KUKA KRL program: EPS_2_251806_MH02A_A_20260213065129.src

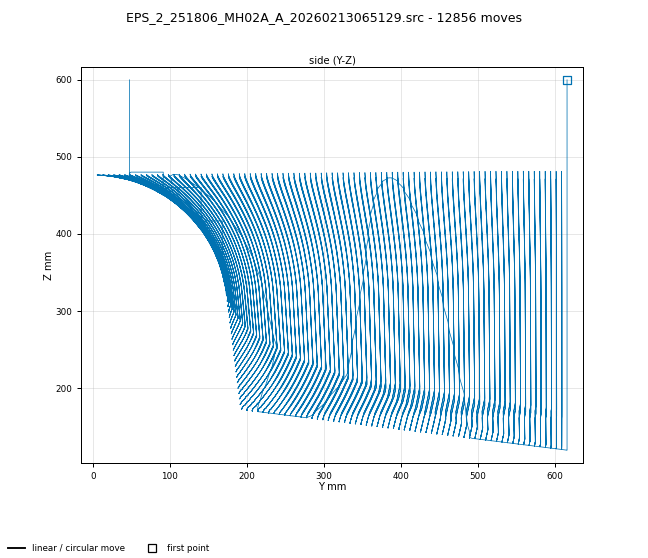
[picture p0: tool path of EPS_2_251806_MH02A_A_20260213065129.src, 12856 of 12858 moves have a stored position in this frame; points joined in program order, loops and branches not executed]
&ACCESS RVP
&REL 4
&COMMENT QRS 19112012
&PARAM EDITMASK = *
DEF PART()
EXT BAS (BAS_COMMAND :IN,REAL :IN )
INT I
BAS (#INITMOV,0 )

;KUKA QRS Post kuka4.cps  Date:22-06-2017 !

File_ID=3031

QRS_PRE_INIT()

;Init var - Until changes are made in qrs_pre_init
Outlet_Square_prg=0
Inlet_1_Square_prg=0
Inlet_2_Square_prg=0
Inlet_3_Square_prg=0
Inlet_4_Square_prg=0
Inlet_5_Square_prg=0

Outlet_1={X 0.000, Y 534.640, Z 332.000, B 0.000, E1 0.000 }
Inlet_1={X 0.000, Y 535.370, Z 322.000, B 0.000, E1 180.000 }
Outlet_1_type=299
Inlet_1_type=299
;QRS#1=Sidecore dimensions
;QRS#2=300-12" PVC SDR 35
;QRS#3=300-12" PVC SDR 35
;QRS#4=
;QRS#5=
;QRS#6=
;QRS#7=
;QRS#8=
;QRS#9=16M PSX
;QRS#10=16M PSX
;QRS#11=
;QRS#12=
;QRS#13=
;QRS#14=
;QRS#15=
;QRS#16=1220x127x762 2,5'
;QRS#17=EPS Height
;QRS#18=481,5
;QRS#19=*
;QRS#20= UPDATED VERSION 22-06-2017
;QRS#21=*
Outlet_Square=0150
Inlet_1_Square=0150
Inlet_2_Square=0
Inlet_3_Square=0
Inlet_4_Square=0
Inlet_5_Square=0
Mill_Square=1
Outlet_Square_Prg=206
Inlet_1_Square_prg=206

QRS_INIT()

$ADVANCE=5

; T1
PTP {E1 173.622,E2 173.622}
PTP {X 0,Y 615.493,A -85,B 0,C 180,E1 173.622,E2 173.622,E3 0,E4 0,E5 0,E6 0}
QRS_SPEED_INIT()
LIN {X 0,Y 615.493,Z 600,A -85,B 0,C 180,E1 173.622,E2 173.622,E3 0,E4 0,E5 0,E6 0} C_VEL
LIN {X 0,Y 615.493,Z 129.502,A -85,B 0,C 180,E1 173.622,E2 173.622} C_VEL
LIN {X 0,Y 615.493,Z 121.323,A -85,B 0,C 180,E1 173.622,E2 173.622} C_VEL
LIN {X 0,Y 615.472,Z 119.323,A -85,B 0,C 180,E1 173.436,E2 173.436} C_VEL
LIN {X 0,Y 615.449,Z 119.317,A -85,B 0,C 180,E1 170.801,E2 170.801} C_VEL
LIN {X 0,Y 615.493,Z 119.316,A -85,B 0,C 180,E1 168.139,E2 168.139} C_VEL
LIN {X 0,Y 615.454,Z 119.321,A -85,B 0,C 180,E1 165.45,E2 165.45} C_VEL
LIN {X 0,Y 615.447,Z 119.321,A -85,B 0,C 180,E1 163.412,E2 163.412} C_VEL
LIN {X 0,Y 615.444,Z 119.32,A -85,B 0,C 180,E1 161.353,E2 161.353} C_VEL
LIN {X 0,Y 615.488,Z 119.314,A -85,B 0,C 180,E1 158.568,E2 158.568} C_VEL
LIN {X 0,Y 615.452,Z 119.322,A -85,B 0,C 180,E1 155.726,E2 155.726} C_VEL
LIN {X 0,Y 615.44,Z 119.321,A -85,B 0,C 180,E1 153.554,E2 153.554} C_VEL
LIN {X 0,Y 615.44,Z 119.319,A -85,B 0,C 180,E1 151.339,E2 151.339} C_VEL
LIN {X 0,Y 615.471,Z 119.316,A -85,B 0,C 180,E1 148.917,E2 148.917} C_VEL
LIN {X 0,Y 615.448,Z 119.322,A -85,B 0,C 180,E1 145.975,E2 145.975} C_VEL
LIN {X 0,Y 615.436,Z 119.32,A -85,B 0,C 180,E1 143.572,E2 143.572} C_VEL
LIN {X 0,Y 615.49,Z 119.316,A -85,B 0,C 180,E1 140.938,E2 140.938} C_VEL
LIN {X 0,Y 615.476,Z 119.325,A -85,B 0,C 180,E1 138.525,E2 138.525} C_VEL
LIN {X 0,Y 615.433,Z 119.322,A -85,B 0,C 180,E1 136.008,E2 136.008} C_VEL
LIN {X 0,Y 615.431,Z 119.321,A -85,B 0,C 180,E1 133.992,E2 133.992} C_VEL
LIN {X 0,Y 615.451,Z 119.319,A -85,B 0,C 180,E1 131.477,E2 131.477} C_VEL
LIN {X 0,Y 615.493,Z 119.325,A -85,B 0,C 180,E1 128.904,E2 128.904} C_VEL
LIN {X 0,Y 615.436,Z 119.323,A -85,B 0,C 180,E1 126.428,E2 126.428} C_VEL
LIN {X 0,Y 615.427,Z 119.322,A -85,B 0,C 180,E1 124.026,E2 124.026} C_VEL
LIN {X 0,Y 615.482,Z 119.326,A -85,B 0,C 180,E1 121.085,E2 121.085} C_VEL
LIN {X 0,Y 615.425,Z 119.323,A -85,B 0,C 180,E1 118.439,E2 118.439} C_VEL
LIN {X 0,Y 615.423,Z 119.323,A -85,B 0,C 180,E1 116.447,E2 116.447} C_VEL
LIN {X 0,Y 615.436,Z 119.322,A -85,B 0,C 180,E1 113.997,E2 113.997} C_VEL
LIN {X 0,Y 615.497,Z 119.53,A -85,B 0,C 180,E1 113.289,E2 113.289} C_VEL
LIN {X 0,Y 615.495,Z 121.309,A -85,B 0,C 180,E1 113.022,E2 113.022} C_VEL
LIN {X 0,Y 615.479,Z 143.31,A -85,B 0,C 180,E1 110.295,E2 110.295} C_VEL
LIN {X 0,Y 615.483,Z 160.451,A -85,B 0,C 180,E1 108.217,E2 108.217} C_VEL
LIN {X 0,Y 615.484,Z 163.048,A -85,B 0,C 180,E1 108.157,E2 108.157} C_VEL
LIN {X 0,Y 615.498,Z 326.22,A -85,B 0,C 180,E1 106.186,E2 106.186} C_VEL
LIN {X 0,Y 615.497,Z 341.617,A -85,B 0,C 180,E1 105.862,E2 105.862} C_VEL
LIN {X 0,Y 615.487,Z 356.978,A -85,B 0,C 180,E1 105.396,E2 105.396} C_VEL
LIN {X 0,Y 615.487,Z 371.662,A -85,B 0,C 180,E1 104.803,E2 104.803} C_VEL
LIN {X 0,Y 615.493,Z 385.63,A -85,B 0,C 180,E1 104.09,E2 104.09} C_VEL
LIN {X 0,Y 615.498,Z 398.491,A -85,B 0,C 180,E1 103.285,E2 103.285} C_VEL
LIN {X 0,Y 615.496,Z 410.744,A -85,B 0,C 180,E1 102.362,E2 102.362} C_VEL
LIN {X 0,Y 615.498,Z 421.898,A -85,B 0,C 180,E1 101.36,E2 101.36} C_VEL
LIN {X 0,Y 615.497,Z 432.703,A -85,B 0,C 180,E1 100.194,E2 100.194} C_VEL
LIN {X 0,Y 615.495,Z 441.685,A -85,B 0,C 180,E1 99.033,E2 99.033} C_VEL
LIN {X 0,Y 615.493,Z 449.119,A -85,B 0,C 180,E1 97.876,E2 97.876} C_VEL
LIN {X 0,Y 615.492,Z 456.052,A -85,B 0,C 180,E1 96.557,E2 96.557} C_VEL
LIN {X 0,Y 615.489,Z 461.498,A -85,B 0,C 180,E1 95.241,E2 95.241} C_VEL
LIN {X 0,Y 615.495,Z 465.619,A -85,B 0,C 180,E1 93.928,E2 93.928} C_VEL
LIN {X 0,Y 615.493,Z 468.525,A -85,B 0,C 180,E1 92.618,E2 92.618} C_VEL
LIN {X 0,Y 615.491,Z 470.276,A -85,B 0,C 180,E1 91.309,E2 91.309} C_VEL
LIN {X 0,Y 615.492,Z 470.884,A -85,B 0,C 180,E1 90,E2 90} C_VEL
LIN {X 0,Y 615.493,Z 470.338,A -85,B 0,C 180,E1 88.691,E2 88.691} C_VEL
LIN {X 0,Y 615.496,Z 468.674,A -85,B 0,C 180,E1 87.382,E2 87.382} C_VEL
LIN {X 0,Y 615.494,Z 465.861,A -85,B 0,C 180,E1 86.072,E2 86.072} C_VEL
LIN {X 0,Y 615.489,Z 461.835,A -85,B 0,C 180,E1 84.759,E2 84.759} C_VEL
LIN {X 0,Y 615.491,Z 456.378,A -85,B 0,C 180,E1 83.42,E2 83.42} C_VEL
LIN {X 0,Y 615.494,Z 449.66,A -85,B 0,C 180,E1 82.124,E2 82.124} C_VEL
LIN {X 0,Y 615.491,Z 441.144,A -85,B 0,C 180,E1 80.801,E2 80.801} C_VEL
LIN {X 0,Y 615.494,Z 432.066,A -85,B 0,C 180,E1 79.639,E2 79.639} C_VEL
LIN {X 0,Y 615.493,Z 422.792,A -85,B 0,C 180,E1 78.64,E2 78.64} C_VEL
LIN {X 0,Y 615.496,Z 410.821,A -85,B 0,C 180,E1 77.554,E2 77.554} C_VEL
LIN {X 0,Y 615.497,Z 398.58,A -85,B 0,C 180,E1 76.631,E2 76.631} C_VEL
LIN {X 0,Y 615.497,Z 385.88,A -85,B 0,C 180,E1 75.834,E2 75.834} C_VEL
LIN {X 0,Y 615.484,Z 371.779,A -85,B 0,C 180,E1 75.113,E2 75.113} C_VEL
LIN {X 0,Y 615.49,Z 357.12,A -85,B 0,C 180,E1 74.52,E2 74.52} C_VEL
LIN {X 0,Y 615.498,Z 342.157,A -85,B 0,C 180,E1 74.062,E2 74.062} C_VEL
LIN {X 0,Y 615.499,Z 326.655,A -85,B 0,C 180,E1 73.732,E2 73.732} C_VEL
LIN {X 0,Y 615.498,Z 214,A -85,B 0,C 180,E1 72.365,E2 72.365} C_VEL
LIN {X 0,Y 615.492,Z 161.034,A -85,B 0,C 180,E1 71.723,E2 71.723} C_VEL
LIN {X 0,Y 615.478,Z 159.241,A -85,B 0,C 180,E1 71.562,E2 71.562} C_VEL
LIN {X 0,Y 615.486,Z 136.234,A -85,B 0,C 180,E1 68.744,E2 68.744} C_VEL
LIN {X 0,Y 615.496,Z 119.705,A -85,B 0,C 180,E1 66.667,E2 66.667} C_VEL
LIN {X 0,Y 615.476,Z 119.33,A -85,B 0,C 180,E1 66.443,E2 66.443} C_VEL
LIN {X 0,Y 615.457,Z 119.324,A -85,B 0,C 180,E1 64.283,E2 64.283} C_VEL
LIN {X 0,Y 615.433,Z 119.324,A -85,B 0,C 180,E1 62.082,E2 62.082} C_VEL
LIN {X 0,Y 615.417,Z 119.324,A -85,B 0,C 180,E1 59.836,E2 59.836} C_VEL
LIN {X 0,Y 615.422,Z 119.324,A -85,B 0,C 180,E1 57.539,E2 57.539} C_VEL
LIN {X 0,Y 615.455,Z 119.325,A -85,B 0,C 180,E1 55.183,E2 55.183} C_VEL
LIN {X 0,Y 615.486,Z 119.322,A -85,B 0,C 180,E1 52.758,E2 52.758} C_VEL
LIN {X 0,Y 615.429,Z 119.322,A -85,B 0,C 180,E1 50.245,E2 50.245} C_VEL
LIN {X 0,Y 615.424,Z 119.323,A -85,B 0,C 180,E1 47.927,E2 47.927} C_VEL
LIN {X 0,Y 615.428,Z 119.323,A -85,B 0,C 180,E1 45.845,E2 45.845} C_VEL
LIN {X 0,Y 615.494,Z 119.325,A -85,B 0,C 180,E1 43.244,E2 43.244} C_VEL
LIN {X 0,Y 615.443,Z 119.32,A -85,B 0,C 180,E1 40.61,E2 40.61} C_VEL
LIN {X 0,Y 615.431,Z 119.322,A -85,B 0,C 180,E1 38.073,E2 38.073} C_VEL
LIN {X 0,Y 615.473,Z 119.324,A -85,B 0,C 180,E1 35.617,E2 35.617} C_VEL
LIN {X 0,Y 615.485,Z 119.319,A -85,B 0,C 180,E1 33.236,E2 33.236} C_VEL
LIN {X 0,Y 615.453,Z 119.318,A -85,B 0,C 180,E1 30.922,E2 30.922} C_VEL
LIN {X 0,Y 615.434,Z 119.321,A -85,B 0,C 180,E1 28.441,E2 28.441} C_VEL
LIN {X 0,Y 615.494,Z 119.321,A -85,B 0,C 180,E1 25.57,E2 25.57} C_VEL
LIN {X 0,Y 615.439,Z 119.319,A -85,B 0,C 180,E1 22.847,E2 22.847} C_VEL
LIN {X 0,Y 615.44,Z 119.321,A -85,B 0,C 180,E1 20.544,E2 20.544} C_VEL
LIN {X 0,Y 615.494,Z 119.326,A -85,B 0,C 180,E1 17.957,E2 17.957} C_VEL
LIN {X 0,Y 615.453,Z 119.317,A -85,B 0,C 180,E1 15.227,E2 15.227} C_VEL
LIN {X 0,Y 615.45,Z 119.317,A -85,B 0,C 180,E1 13.202,E2 13.202} C_VEL
LIN {X 0,Y 615.442,Z 119.32,A -85,B 0,C 180,E1 10.865,E2 10.865} C_VEL
LIN {X 0,Y 615.463,Z 119.322,A -85,B 0,C 180,E1 8.537,E2 8.537} C_VEL
LIN {X 0,Y 615.499,Z 119.313,A -85,B 0,C 180,E1 5.899,E2 5.899} C_VEL
LIN {X 0,Y 615.447,Z 119.317,A -85,B 0,C 180,E1 3.273,E2 3.273} C_VEL
LIN {X 0,Y 615.474,Z 119.323,A -85,B 0,C 180,E1 0.654,E2 0.654} C_VEL
LIN {X 0,Y 615.499,Z 119.311,A -85,B 0,C 180,E1 -1.963,E2 -1.963} C_VEL
LIN {X 0,Y 615.45,Z 119.317,A -85,B 0,C 180,E1 -4.585,E2 -4.585} C_VEL
LIN {X 0,Y 615.48,Z 119.325,A -85,B 0,C 180,E1 -7.216,E2 -7.216} C_VEL
LIN {X 0,Y 615.49,Z 119.31,A -85,B 0,C 180,E1 -9.862,E2 -9.862} C_VEL
LIN {X 0,Y 615.453,Z 119.318,A -85,B 0,C 180,E1 -12.531,E2 -12.531} C_VEL
LIN {X 0,Y 615.494,Z 119.322,A -85,B 0,C 180,E1 -15.226,E2 -15.226} C_VEL
LIN {X 0,Y 615.466,Z 119.313,A -85,B 0,C 180,E1 -17.958,E2 -17.958} C_VEL
LIN {X 0,Y 615.463,Z 119.321,A -85,B 0,C 180,E1 -20.55,E2 -20.55} C_VEL
LIN {X 0,Y 615.485,Z 119.327,A -85,B 0,C 180,E1 -22.845,E2 -22.845} C_VEL
LIN {X 0,Y 615.473,Z 119.311,A -85,B 0,C 180,E1 -25.716,E2 -25.716} C_VEL
LIN {X 0,Y 615.469,Z 119.323,A -85,B 0,C 180,E1 -28.447,E2 -28.447} C_VEL
LIN {X 0,Y 615.491,Z 119.313,A -85,B 0,C 180,E1 -31.086,E2 -31.086} C_VEL
LIN {X 0,Y 615.475,Z 119.311,A -85,B 0,C 180,E1 -33.532,E2 -33.532} C_VEL
LIN {X 0,Y 615.462,Z 119.316,A -85,B 0,C 180,E1 -35.83,E2 -35.83} C_VEL
LIN {X 0,Y 615.469,Z 119.32,A -85,B 0,C 180,E1 -38.07,E2 -38.07} C_VEL
LIN {X 0,Y 615.49,Z 119.319,A -85,B 0,C 180,E1 -40.606,E2 -40.606} C_VEL
LIN {X 0,Y 615.481,Z 119.309,A -85,B 0,C 180,E1 -43.245,E2 -43.245} C_VEL
LIN {X 0,Y 615.478,Z 119.323,A -85,B 0,C 180,E1 -46.003,E2 -46.003} C_VEL
LIN {X 0,Y 615.487,Z 119.309,A -85,B 0,C 180,E1 -48.905,E2 -48.905} C_VEL
LIN {X 0,Y 615.48,Z 119.31,A -85,B 0,C 180,E1 -51.095,E2 -51.095} C_VEL
LIN {X 0,Y 615.471,Z 119.318,A -85,B 0,C 180,E1 -53.574,E2 -53.574} C_VEL
LIN {X 0,Y 615.486,Z 119.312,A -85,B 0,C 180,E1 -56.466,E2 -56.466} C_VEL
LIN {X 0,Y 615.472,Z 119.313,A -85,B 0,C 180,E1 -59.079,E2 -59.079} C_VEL
LIN {X 0,Y 615.48,Z 119.322,A -85,B 0,C 180,E1 -61.551,E2 -61.551} C_VEL
LIN {X 0,Y 615.487,Z 119.309,A -85,B 0,C 180,E1 -64.431,E2 -64.431} C_VEL
LIN {X 0,Y 615.497,Z 119.517,A -85,B 0,C 180,E1 -65.761,E2 -65.761} C_VEL
LIN {X 0,Y 615.468,Z 138.379,A -85,B 0,C 180,E1 -68.039,E2 -68.039} C_VEL
LIN {X 0,Y 615.469,Z 162.221,A -85,B 0,C 180,E1 -70.835,E2 -70.835} C_VEL
LIN {X 0,Y 615.495,Z 170.191,A -85,B 0,C 180,E1 -71.741,E2 -71.741} C_VEL
LIN {X 0,Y 615.49,Z 178.359,A -85,B 0,C 180,E1 -71.862,E2 -71.862} C_VEL
LIN {X 0,Y 615.498,Z 335.92,A -85,B 0,C 180,E1 -73.764,E2 -73.764} C_VEL
LIN {X 0,Y 615.497,Z 351.711,A -85,B 0,C 180,E1 -74.095,E2 -74.095} C_VEL
LIN {X 0,Y 615.489,Z 367.049,A -85,B 0,C 180,E1 -74.562,E2 -74.562} C_VEL
LIN {X 0,Y 615.485,Z 380.752,A -85,B 0,C 180,E1 -75.113,E2 -75.113} C_VEL
LIN {X 0,Y 615.493,Z 395.046,A -85,B 0,C 180,E1 -75.833,E2 -75.833} C_VEL
LIN {X 0,Y 615.497,Z 407.898,A -85,B 0,C 180,E1 -76.631,E2 -76.631} C_VEL
LIN {X 0,Y 615.495,Z 420.254,A -85,B 0,C 180,E1 -77.554,E2 -77.554} C_VEL
LIN {X 0,Y 615.496,Z 430.606,A -85,B 0,C 180,E1 -78.473,E2 -78.473} C_VEL
LIN {X 0,Y 615.494,Z 440.184,A -85,B 0,C 180,E1 -79.473,E2 -79.473} C_VEL
LIN {X 0,Y 615.494,Z 449.577,A -85,B 0,C 180,E1 -80.636,E2 -80.636} C_VEL
LIN {X 0,Y 615.494,Z 457.381,A -85,B 0,C 180,E1 -81.794,E2 -81.794} C_VEL
LIN {X 0,Y 615.494,Z 464.609,A -85,B 0,C 180,E1 -83.102,E2 -83.102} C_VEL
LIN {X 0,Y 615.499,Z 470.436,A -85,B 0,C 180,E1 -84.43,E2 -84.43} C_VEL
LIN {X 0,Y 615.491,Z 473.86,A -85,B 0,C 180,E1 -85.415,E2 -85.415} C_VEL
LIN {X 0,Y 615.493,Z 477.318,A -85,B 0,C 180,E1 -86.727,E2 -86.727} C_VEL
LIN {X 0,Y 615.5,Z 479.593,A -85,B 0,C 180,E1 -88.037,E2 -88.037} C_VEL
LIN {X 0,Y 615.491,Z 480.741,A -85,B 0,C 180,E1 -89.346,E2 -89.346} C_VEL
LIN {X 0,Y 615.491,Z 480.741,A -85,B 0,C 180,E1 -90.654,E2 -90.654} C_VEL
LIN {X 0,Y 615.5,Z 479.593,A -85,B 0,C 180,E1 -91.963,E2 -91.963} C_VEL
LIN {X 0,Y 615.493,Z 477.318,A -85,B 0,C 180,E1 -93.273,E2 -93.273} C_VEL
LIN {X 0,Y 615.491,Z 473.86,A -85,B 0,C 180,E1 -94.585,E2 -94.585} C_VEL
LIN {X 0,Y 615.499,Z 469.142,A -85,B 0,C 180,E1 -95.898,E2 -95.898} C_VEL
LIN {X 0,Y 615.492,Z 463.03,A -85,B 0,C 180,E1 -97.216,E2 -97.216} C_VEL
LIN {X 0,Y 615.493,Z 455.332,A -85,B 0,C 180,E1 -98.537,E2 -98.537} C_VEL
LIN {X 0,Y 615.495,Z 447.114,A -85,B 0,C 180,E1 -99.696,E2 -99.696} C_VEL
LIN {X 0,Y 615.496,Z 436.899,A -85,B 0,C 180,E1 -100.892,E2 -100.892} C_VEL
LIN {X 0,Y 615.496,Z 427.067,A -85,B 0,C 180,E1 -101.861,E2 -101.861} C_VEL
LIN {X 0,Y 615.497,Z 414.947,A -85,B 0,C 180,E1 -102.865,E2 -102.865} C_VEL
LIN {X 0,Y 615.498,Z 402.797,A -85,B 0,C 180,E1 -103.706,E2 -103.706} C_VEL
LIN {X 0,Y 615.48,Z 389.379,A -85,B 0,C 180,E1 -104.473,E2 -104.473} C_VEL
LIN {X 0,Y 615.494,Z 374.847,A -85,B 0,C 180,E1 -105.141,E2 -105.141} C_VEL
LIN {X 0,Y 615.495,Z 360.615,A -85,B 0,C 180,E1 -105.65,E2 -105.65} C_VEL
LIN {X 0,Y 615.5,Z 346.077,A -85,B 0,C 180,E1 -106.037,E2 -106.037} C_VEL
LIN {X 0,Y 615.498,Z 331.292,A -85,B 0,C 180,E1 -106.301,E2 -106.301} C_VEL
LIN {X 0,Y 615.494,Z 170.613,A -85,B 0,C 180,E1 -108.238,E2 -108.238} C_VEL
LIN {X 0,Y 615.485,Z 168.467,A -85,B 0,C 180,E1 -108.44,E2 -108.44} C_VEL
LIN {X 0,Y 615.486,Z 144.341,A -85,B 0,C 180,E1 -111.256,E2 -111.256} C_VEL
LIN {X 0,Y 615.498,Z 121.176,A -85,B 0,C 180,E1 -114.011,E2 -114.011} C_VEL
LIN {X 0,Y 615.495,Z 119.429,A -85,B 0,C 180,E1 -114.272,E2 -114.272} C_VEL
LIN {X 0,Y 615.474,Z 119.312,A -85,B 0,C 180,E1 -117.043,E2 -117.043} C_VEL
LIN {X 0,Y 615.484,Z 119.316,A -85,B 0,C 180,E1 -119.794,E2 -119.794} C_VEL
LIN {X 0,Y 615.476,Z 119.319,A -85,B 0,C 180,E1 -122.458,E2 -122.458} C_VEL
LIN {X 0,Y 615.471,Z 119.313,A -85,B 0,C 180,E1 -124.816,E2 -124.816} C_VEL
LIN {X 0,Y 615.494,Z 119.308,A -85,B 0,C 180,E1 -127.242,E2 -127.242} C_VEL
LIN {X 0,Y 615.484,Z 119.322,A -85,B 0,C 180,E1 -130.089,E2 -130.089} C_VEL
LIN {X 0,Y 615.468,Z 119.317,A -85,B 0,C 180,E1 -132.355,E2 -132.355} C_VEL
LIN {X 0,Y 615.491,Z 119.309,A -85,B 0,C 180,E1 -135.068,E2 -135.068} C_VEL
LIN {X 0,Y 615.479,Z 119.322,A -85,B 0,C 180,E1 -137.921,E2 -137.921} C_VEL
LIN {X 0,Y 615.464,Z 119.316,A -85,B 0,C 180,E1 -140.248,E2 -140.248} C_VEL
LIN {X 0,Y 615.49,Z 119.313,A -85,B 0,C 180,E1 -143.063,E2 -143.063} C_VEL
LIN {X 0,Y 615.464,Z 119.318,A -85,B 0,C 180,E1 -145.977,E2 -145.977} C_VEL
LIN {X 0,Y 615.465,Z 119.313,A -85,B 0,C 180,E1 -148.313,E2 -148.313} C_VEL
LIN {X 0,Y 615.486,Z 119.31,A -85,B 0,C 180,E1 -150.594,E2 -150.594} C_VEL
LIN {X 0,Y 615.472,Z 119.321,A -85,B 0,C 180,E1 -153.555,E2 -153.555} C_VEL
LIN {X 0,Y 615.461,Z 119.315,A -85,B 0,C 180,E1 -155.998,E2 -155.998} C_VEL
LIN {X 0,Y 615.496,Z 119.31,A -85,B 0,C 180,E1 -158.568,E2 -158.568} C_VEL
LIN {X 0,Y 615.466,Z 119.321,A -85,B 0,C 180,E1 -161.402,E2 -161.402} C_VEL
LIN {X 0,Y 615.474,Z 119.311,A -85,B 0,C 180,E1 -164.095,E2 -164.095} C_VEL
LIN {X 0,Y 615.493,Z 119.324,A -85,B 0,C 180,E1 -166.799,E2 -166.799} C_VEL
LIN {X 0,Y 615.454,Z 119.318,A -85,B 0,C 180,E1 -169.473,E2 -169.473} C_VEL
LIN {X 0,Y 615.484,Z 119.312,A -85,B 0,C 180,E1 -172.124,E2 -172.124} C_VEL
LIN {X 0,Y 615.487,Z 119.324,A -85,B 0,C 180,E1 -174.759,E2 -174.759} C_VEL
LIN {X 0,Y 615.452,Z 119.317,A -85,B 0,C 180,E1 -177.382,E2 -177.382} C_VEL
LIN {X 0,Y 615.487,Z 119.313,A -85,B 0,C 180,E1 -180,E2 -180} C_VEL
LIN {X 0,Y 615.478,Z 119.323,A -85,B 0,C 180,E1 -182.618,E2 -182.618} C_VEL
LIN {X 0,Y 615.448,Z 119.317,A -85,B 0,C 180,E1 -185.242,E2 -185.242} C_VEL
LIN {X 0,Y 615.472,Z 119.323,A -85,B 0,C 180,E1 -186.564,E2 -186.564} C_VEL
LIN {X 0,Y 614.779,Z 119.464,A -85,B 0,C 180,E1 -187.11,E2 -187.11} C_VEL
LIN {X 0,Y 611.93,Z 119.885,A -85,B 0,C 180,E1 -187.996,E2 -187.996} C_VEL
LIN {X 0,Y 609.543,Z 120.19,A -85,B 0,C 180,E1 -188.709,E2 -188.709} C_VEL
LIN {X 0,Y 608.523,Z 120.305,A -85,B 0,C 180,E1 -189.258,E2 -189.258} C_VEL
LIN {X 0,Y 608.441,Z 120.314,A -85,B 0,C 180,E1 -189.444,E2 -189.444} C_VEL
LIN {X 0,Y 608.461,Z 120.319,A -85,B 0,C 180,E1 -192,E2 -192} C_VEL
LIN {X 0,Y 608.418,Z 120.318,A -85,B 0,C 180,E1 -194.722,E2 -194.722} C_VEL
LIN {X 0,Y 608.421,Z 120.317,A -85,B 0,C 180,E1 -196.785,E2 -196.785} C_VEL
LIN {X 0,Y 608.443,Z 120.318,A -85,B 0,C 180,E1 -199.571,E2 -199.571} C_VEL
LIN {X 0,Y 608.431,Z 120.317,A -85,B 0,C 180,E1 -202.469,E2 -202.469} C_VEL
LIN {X 0,Y 608.425,Z 120.316,A -85,B 0,C 180,E1 -204.572,E2 -204.572} C_VEL
LIN {X 0,Y 608.464,Z 120.314,A -85,B 0,C 180,E1 -207.204,E2 -207.204} C_VEL
LIN {X 0,Y 608.435,Z 120.32,A -85,B 0,C 180,E1 -209.966,E2 -209.966} C_VEL
LIN {X 0,Y 608.421,Z 120.316,A -85,B 0,C 180,E1 -212.516,E2 -212.516} C_VEL
LIN {X 0,Y 608.43,Z 120.322,A -85,B 0,C 180,E1 -215.279,E2 -215.279} C_VEL
LIN {X 0,Y 608.445,Z 120.318,A -85,B 0,C 180,E1 -217.748,E2 -217.748} C_VEL
LIN {X 0,Y 608.405,Z 120.318,A -85,B 0,C 180,E1 -220.324,E2 -220.324} C_VEL
LIN {X 0,Y 608.447,Z 120.318,A -85,B 0,C 180,E1 -222.96,E2 -222.96} C_VEL
LIN {X 0,Y 608.416,Z 120.319,A -85,B 0,C 180,E1 -225.74,E2 -225.74} C_VEL
LIN {X 0,Y 608.415,Z 120.318,A -85,B 0,C 180,E1 -227.935,E2 -227.935} C_VEL
LIN {X 0,Y 608.439,Z 120.319,A -85,B 0,C 180,E1 -230.706,E2 -230.706} C_VEL
LIN {X 0,Y 608.453,Z 120.322,A -85,B 0,C 180,E1 -233.085,E2 -233.085} C_VEL
LIN {X 0,Y 608.433,Z 120.317,A -85,B 0,C 180,E1 -235.528,E2 -235.528} C_VEL
LIN {X 0,Y 608.418,Z 120.317,A -85,B 0,C 180,E1 -237.903,E2 -237.903} C_VEL
LIN {X 0,Y 608.43,Z 120.317,A -85,B 0,C 180,E1 -240.218,E2 -240.218} C_VEL
LIN {X 0,Y 608.47,Z 120.32,A -85,B 0,C 180,E1 -242.795,E2 -242.795} C_VEL
LIN {X 0,Y 608.411,Z 120.32,A -85,B 0,C 180,E1 -245.427,E2 -245.427} C_VEL
LIN {X 0,Y 608.492,Z 120.487,A -85,B 0,C 180,E1 -246.562,E2 -246.562} C_VEL
LIN {X 0,Y 608.611,Z 124.155,A -85,B 0,C 180,E1 -247.062,E2 -247.062} C_VEL
LIN {X 0,Y 608.564,Z 145.448,A -85,B 0,C 180,E1 -249.729,E2 -249.729} C_VEL
LIN {X 0,Y 608.538,Z 160.451,A -85,B 0,C 180,E1 -251.568,E2 -251.568} C_VEL
LIN {X 0,Y 608.757,Z 163.093,A -85,B 0,C 180,E1 -251.635,E2 -251.635} C_VEL
LIN {X 0,Y 608.699,Z 326.277,A -85,B 0,C 180,E1 -253.629,E2 -253.629} C_VEL
LIN {X 0,Y 608.67,Z 341.638,A -85,B 0,C 180,E1 -253.955,E2 -253.955} C_VEL
LIN {X 0,Y 608.619,Z 356.993,A -85,B 0,C 180,E1 -254.426,E2 -254.426} C_VEL
LIN {X 0,Y 608.586,Z 371.674,A -85,B 0,C 180,E1 -255.026,E2 -255.026} C_VEL
LIN {X 0,Y 608.571,Z 385.441,A -85,B 0,C 180,E1 -255.735,E2 -255.735} C_VEL
LIN {X 0,Y 608.548,Z 398.544,A -85,B 0,C 180,E1 -256.56,E2 -256.56} C_VEL
LIN {X 0,Y 608.505,Z 410.84,A -85,B 0,C 180,E1 -257.493,E2 -257.493} C_VEL
LIN {X 0,Y 608.498,Z 422.05,A -85,B 0,C 180,E1 -258.508,E2 -258.508} C_VEL
LIN {X 0,Y 608.477,Z 432.935,A -85,B 0,C 180,E1 -259.687,E2 -259.687} C_VEL
LIN {X 0,Y 608.469,Z 441.984,A -85,B 0,C 180,E1 -260.862,E2 -260.862} C_VEL
LIN {X 0,Y 608.456,Z 449.48,A -85,B 0,C 180,E1 -262.033,E2 -262.033} C_VEL
LIN {X 0,Y 608.445,Z 456.629,A -85,B 0,C 180,E1 -263.397,E2 -263.397} C_VEL
LIN {X 0,Y 608.435,Z 461.994,A -85,B 0,C 180,E1 -264.698,E2 -264.698} C_VEL
LIN {X 0,Y 608.431,Z 466.167,A -85,B 0,C 180,E1 -266.026,E2 -266.026} C_VEL
LIN {X 0,Y 608.421,Z 469.11,A -85,B 0,C 180,E1 -267.352,E2 -267.352} C_VEL
LIN {X 0,Y 608.444,Z 470.88,A -85,B 0,C 180,E1 -268.676,E2 -268.676} C_VEL
LIN {X 0,Y 608.432,Z 471.495,A -85,B 0,C 180,E1 -270,E2 -270} C_VEL
LIN {X 0,Y 608.445,Z 470.944,A -85,B 0,C 180,E1 -271.324,E2 -271.324} C_VEL
LIN {X 0,Y 608.424,Z 469.259,A -85,B 0,C 180,E1 -272.648,E2 -272.648} C_VEL
LIN {X 0,Y 608.431,Z 466.408,A -85,B 0,C 180,E1 -273.974,E2 -273.974} C_VEL
LIN {X 0,Y 608.435,Z 462.328,A -85,B 0,C 180,E1 -275.302,E2 -275.302} C_VEL
LIN {X 0,Y 608.446,Z 456.921,A -85,B 0,C 180,E1 -276.633,E2 -276.633} C_VEL
LIN {X 0,Y 608.457,Z 450.022,A -85,B 0,C 180,E1 -277.967,E2 -277.967} C_VEL
LIN {X 0,Y 608.466,Z 442.591,A -85,B 0,C 180,E1 -279.138,E2 -279.138} C_VEL
LIN {X 0,Y 608.476,Z 433.662,A -85,B 0,C 180,E1 -280.313,E2 -280.313} C_VEL
LIN {X 0,Y 608.495,Z 422.946,A -85,B 0,C 180,E1 -281.492,E2 -281.492} C_VEL
LIN {X 0,Y 608.513,Z 410.905,A -85,B 0,C 180,E1 -282.591,E2 -282.591} C_VEL
LIN {X 0,Y 608.543,Z 398.616,A -85,B 0,C 180,E1 -283.525,E2 -283.525} C_VEL
LIN {X 0,Y 608.585,Z 385.673,A -85,B 0,C 180,E1 -284.342,E2 -284.342} C_VEL
LIN {X 0,Y 608.586,Z 371.767,A -85,B 0,C 180,E1 -285.06,E2 -285.06} C_VEL
LIN {X 0,Y 608.645,Z 357.103,A -85,B 0,C 180,E1 -285.659,E2 -285.659} C_VEL
LIN {X 0,Y 608.67,Z 341.514,A -85,B 0,C 180,E1 -286.138,E2 -286.138} C_VEL
LIN {X 0,Y 608.696,Z 326.113,A -85,B 0,C 180,E1 -286.464,E2 -286.464} C_VEL
LIN {X 0,Y 608.684,Z 161.463,A -85,B 0,C 180,E1 -288.479,E2 -288.479} C_VEL
LIN {X 0,Y 608.548,Z 160.131,A -85,B 0,C 180,E1 -288.552,E2 -288.552} C_VEL
LIN {X 0,Y 608.573,Z 137.649,A -85,B 0,C 180,E1 -291.332,E2 -291.332} C_VEL
LIN {X 0,Y 608.53,Z 120.73,A -85,B 0,C 180,E1 -293.47,E2 -293.47} C_VEL
LIN {X 0,Y 608.437,Z 120.339,A -85,B 0,C 180,E1 -293.665,E2 -293.665} C_VEL
LIN {X 0,Y 608.404,Z 120.32,A -85,B 0,C 180,E1 -296.038,E2 -296.038} C_VEL
LIN {X 0,Y 608.387,Z 120.321,A -85,B 0,C 180,E1 -298.27,E2 -298.27} C_VEL
LIN {X 0,Y 608.406,Z 120.319,A -85,B 0,C 180,E1 -300.548,E2 -300.548} C_VEL
LIN {X 0,Y 608.43,Z 120.321,A -85,B 0,C 180,E1 -302.881,E2 -302.881} C_VEL
LIN {X 0,Y 608.412,Z 120.325,A -85,B 0,C 180,E1 -305.28,E2 -305.28} C_VEL
LIN {X 0,Y 608.429,Z 120.317,A -85,B 0,C 180,E1 -307.749,E2 -307.749} C_VEL
LIN {X 0,Y 608.403,Z 120.32,A -85,B 0,C 180,E1 -310.323,E2 -310.323} C_VEL
LIN {X 0,Y 608.447,Z 120.323,A -85,B 0,C 180,E1 -312.961,E2 -312.961} C_VEL
LIN {X 0,Y 608.407,Z 120.318,A -85,B 0,C 180,E1 -315.741,E2 -315.741} C_VEL
LIN {X 0,Y 608.411,Z 120.318,A -85,B 0,C 180,E1 -317.934,E2 -317.934} C_VEL
LIN {X 0,Y 608.437,Z 120.325,A -85,B 0,C 180,E1 -320.707,E2 -320.707} C_VEL
LIN {X 0,Y 608.436,Z 120.318,A -85,B 0,C 180,E1 -323.084,E2 -323.084} C_VEL
LIN {X 0,Y 608.429,Z 120.315,A -85,B 0,C 180,E1 -325.528,E2 -325.528} C_VEL
LIN {X 0,Y 608.432,Z 120.316,A -85,B 0,C 180,E1 -327.903,E2 -327.903} C_VEL
LIN {X 0,Y 608.457,Z 120.319,A -85,B 0,C 180,E1 -330.22,E2 -330.22} C_VEL
LIN {X 0,Y 608.409,Z 120.318,A -85,B 0,C 180,E1 -333.224,E2 -333.224} C_VEL
LIN {X 0,Y 608.42,Z 120.317,A -85,B 0,C 180,E1 -335.427,E2 -335.427} C_VEL
LIN {X 0,Y 608.46,Z 120.32,A -85,B 0,C 180,E1 -338.308,E2 -338.308} C_VEL
LIN {X 0,Y 608.434,Z 120.315,A -85,B 0,C 180,E1 -341.13,E2 -341.13} C_VEL
LIN {X 0,Y 608.454,Z 120.321,A -85,B 0,C 180,E1 -343.906,E2 -343.906} C_VEL
LIN {X 0,Y 608.44,Z 120.315,A -85,B 0,C 180,E1 -346.643,E2 -346.643} C_VEL
LIN {X 0,Y 608.432,Z 120.318,A -85,B 0,C 180,E1 -349.35,E2 -349.35} C_VEL
LIN {X 0,Y 608.478,Z 120.315,A -85,B 0,C 180,E1 -352.033,E2 -352.033} C_VEL
LIN {X 0,Y 608.431,Z 120.315,A -85,B 0,C 180,E1 -354.698,E2 -354.698} C_VEL
LIN {X 0,Y 608.463,Z 120.317,A -85,B 0,C 180,E1 -357.352,E2 -357.352} C_VEL
LIN {X 0,Y 608.477,Z 120.313,A -85,B 0,C 180,E1 -360,E2 -360} C_VEL
LIN {X 0,Y 608.443,Z 120.314,A -85,B 0,C 180,E1 -362.648,E2 -362.648} C_VEL
LIN {X 0,Y 608.463,Z 120.32,A -85,B 0,C 180,E1 -365.302,E2 -365.302} C_VEL
LIN {X 0,Y 608.472,Z 120.311,A -85,B 0,C 180,E1 -367.967,E2 -367.967} C_VEL
LIN {X 0,Y 608.437,Z 120.316,A -85,B 0,C 180,E1 -370.65,E2 -370.65} C_VEL
LIN {X 0,Y 608.468,Z 120.318,A -85,B 0,C 180,E1 -373.356,E2 -373.356} C_VEL
LIN {X 0,Y 608.442,Z 120.314,A -85,B 0,C 180,E1 -376.094,E2 -376.094} C_VEL
LIN {X 0,Y 608.45,Z 120.321,A -85,B 0,C 180,E1 -378.87,E2 -378.87} C_VEL
LIN {X 0,Y 608.464,Z 120.312,A -85,B 0,C 180,E1 -381.692,E2 -381.692} C_VEL
LIN {X 0,Y 608.443,Z 120.32,A -85,B 0,C 180,E1 -384.571,E2 -384.571} C_VEL
LIN {X 0,Y 608.484,Z 120.312,A -85,B 0,C 180,E1 -387.208,E2 -387.208} C_VEL
LIN {X 0,Y 608.446,Z 120.314,A -85,B 0,C 180,E1 -389.968,E2 -389.968} C_VEL
LIN {X 0,Y 608.457,Z 120.317,A -85,B 0,C 180,E1 -392.879,E2 -392.879} C_VEL
LIN {X 0,Y 608.435,Z 120.315,A -85,B 0,C 180,E1 -395.278,E2 -395.278} C_VEL
LIN {X 0,Y 608.459,Z 120.313,A -85,B 0,C 180,E1 -397.747,E2 -397.747} C_VEL
LIN {X 0,Y 608.446,Z 120.323,A -85,B 0,C 180,E1 -400.328,E2 -400.328} C_VEL
LIN {X 0,Y 608.47,Z 120.311,A -85,B 0,C 180,E1 -403.309,E2 -403.309} C_VEL
LIN {X 0,Y 608.465,Z 120.32,A -85,B 0,C 180,E1 -406.13,E2 -406.13} C_VEL
LIN {X 0,Y 608.457,Z 120.313,A -85,B 0,C 180,E1 -408.823,E2 -408.823} C_VEL
LIN {X 0,Y 608.465,Z 120.312,A -85,B 0,C 180,E1 -411.412,E2 -411.412} C_VEL
LIN {X 0,Y 608.447,Z 120.323,A -85,B 0,C 180,E1 -413.954,E2 -413.954} C_VEL
LIN {X 0,Y 608.467,Z 120.314,A -85,B 0,C 180,E1 -416.329,E2 -416.329} C_VEL
LIN {X 0,Y 608.447,Z 120.313,A -85,B 0,C 180,E1 -418.732,E2 -418.732} C_VEL
LIN {X 0,Y 608.465,Z 120.315,A -85,B 0,C 180,E1 -421.381,E2 -421.381} C_VEL
LIN {X 0,Y 608.446,Z 120.321,A -85,B 0,C 180,E1 -423.964,E2 -423.964} C_VEL
LIN {X 0,Y 608.505,Z 120.443,A -85,B 0,C 180,E1 -425.586,E2 -425.586} C_VEL
LIN {X 0,Y 608.648,Z 129.437,A -85,B 0,C 180,E1 -426.704,E2 -426.704} C_VEL
LIN {X 0,Y 608.545,Z 151.172,A -85,B 0,C 180,E1 -429.302,E2 -429.302} C_VEL
LIN {X 0,Y 608.579,Z 170.183,A -85,B 0,C 180,E1 -431.526,E2 -431.526} C_VEL
LIN {X 0,Y 608.761,Z 173.339,A -85,B 0,C 180,E1 -431.593,E2 -431.593} C_VEL
LIN {X 0,Y 608.692,Z 335.919,A -85,B 0,C 180,E1 -433.578,E2 -433.578} C_VEL
LIN {X 0,Y 608.657,Z 351.709,A -85,B 0,C 180,E1 -433.911,E2 -433.911} C_VEL
LIN {X 0,Y 608.631,Z 367.047,A -85,B 0,C 180,E1 -434.384,E2 -434.384} C_VEL
LIN {X 0,Y 608.6,Z 380.756,A -85,B 0,C 180,E1 -434.94,E2 -434.94} C_VEL
LIN {X 0,Y 608.574,Z 394.236,A -85,B 0,C 180,E1 -435.624,E2 -435.624} C_VEL
LIN {X 0,Y 608.554,Z 406.664,A -85,B 0,C 180,E1 -436.39,E2 -436.39} C_VEL
LIN {X 0,Y 608.528,Z 419.282,A -85,B 0,C 180,E1 -437.324,E2 -437.324} C_VEL
LIN {X 0,Y 608.498,Z 430.747,A -85,B 0,C 180,E1 -438.339,E2 -438.339} C_VEL
LIN {X 0,Y 608.475,Z 440.388,A -85,B 0,C 180,E1 -439.35,E2 -439.35} C_VEL
LIN {X 0,Y 608.477,Z 449.853,A -85,B 0,C 180,E1 -440.527,E2 -440.527} C_VEL
LIN {X 0,Y 608.456,Z 457.729,A -85,B 0,C 180,E1 -441.698,E2 -441.698} C_VEL
LIN {X 0,Y 608.439,Z 465.087,A -85,B 0,C 180,E1 -443.034,E2 -443.034} C_VEL
LIN {X 0,Y 608.451,Z 470.923,A -85,B 0,C 180,E1 -444.366,E2 -444.366} C_VEL
LIN {X 0,Y 608.427,Z 474.383,A -85,B 0,C 180,E1 -445.362,E2 -445.362} C_VEL
LIN {X 0,Y 608.421,Z 477.885,A -85,B 0,C 180,E1 -446.689,E2 -446.689} C_VEL
LIN {X 0,Y 608.444,Z 480.191,A -85,B 0,C 180,E1 -448.014,E2 -448.014} C_VEL
LIN {X 0,Y 608.434,Z 481.35,A -85,B 0,C 180,E1 -449.338,E2 -449.338} C_VEL
LIN {X 0,Y 608.434,Z 481.35,A -85,B 0,C 180,E1 -450.662,E2 -450.662} C_VEL
LIN {X 0,Y 608.444,Z 480.191,A -85,B 0,C 180,E1 -451.986,E2 -451.986} C_VEL
LIN {X 0,Y 608.421,Z 477.885,A -85,B 0,C 180,E1 -453.311,E2 -453.311} C_VEL
LIN {X 0,Y 608.427,Z 474.383,A -85,B 0,C 180,E1 -454.638,E2 -454.638} C_VEL
LIN {X 0,Y 608.437,Z 469.608,A -85,B 0,C 180,E1 -455.967,E2 -455.967} C_VEL
LIN {X 0,Y 608.456,Z 463.426,A -85,B 0,C 180,E1 -457.299,E2 -457.299} C_VEL
LIN {X 0,Y 608.467,Z 455.654,A -85,B 0,C 180,E1 -458.636,E2 -458.636} C_VEL
LIN {X 0,Y 608.471,Z 447.37,A -85,B 0,C 180,E1 -459.809,E2 -459.809} C_VEL
LIN {X 0,Y 608.492,Z 436.652,A -85,B 0,C 180,E1 -461.063,E2 -461.063} C_VEL
LIN {X 0,Y 608.522,Z 425.274,A -85,B 0,C 180,E1 -462.168,E2 -462.168} C_VEL
LIN {X 0,Y 608.547,Z 413.854,A -85,B 0,C 180,E1 -463.1,E2 -463.1} C_VEL
LIN {X 0,Y 608.563,Z 401.447,A -85,B 0,C 180,E1 -463.95,E2 -463.95} C_VEL
LIN {X 0,Y 608.565,Z 387.859,A -85,B 0,C 180,E1 -464.718,E2 -464.718} C_VEL
LIN {X 0,Y 608.609,Z 373.791,A -85,B 0,C 180,E1 -465.359,E2 -465.359} C_VEL
LIN {X 0,Y 608.645,Z 359.3,A -85,B 0,C 180,E1 -465.874,E2 -465.874} C_VEL
LIN {X 0,Y 608.676,Z 343.926,A -85,B 0,C 180,E1 -466.272,E2 -466.272} C_VEL
LIN {X 0,Y 608.703,Z 328.269,A -85,B 0,C 180,E1 -466.531,E2 -466.531} C_VEL
LIN {X 0,Y 608.681,Z 171.016,A -85,B 0,C 180,E1 -468.44,E2 -468.44} C_VEL
LIN {X 0,Y 608.547,Z 169.92,A -85,B 0,C 180,E1 -468.495,E2 -468.495} C_VEL
LIN {X 0,Y 608.588,Z 147.322,A -85,B 0,C 180,E1 -471.154,E2 -471.154} C_VEL
LIN {X 0,Y 608.67,Z 124.966,A -85,B 0,C 180,E1 -473.836,E2 -473.836} C_VEL
LIN {X 0,Y 608.474,Z 120.398,A -85,B 0,C 180,E1 -474.431,E2 -474.431} C_VEL
LIN {X 0,Y 608.474,Z 120.31,A -85,B 0,C 180,E1 -477.206,E2 -477.206} C_VEL
LIN {X 0,Y 608.47,Z 120.317,A -85,B 0,C 180,E1 -479.972,E2 -479.972} C_VEL
LIN {X 0,Y 608.454,Z 120.313,A -85,B 0,C 180,E1 -482.88,E2 -482.88} C_VEL
LIN {X 0,Y 608.435,Z 120.315,A -85,B 0,C 180,E1 -485.278,E2 -485.278} C_VEL
LIN {X 0,Y 608.47,Z 120.317,A -85,B 0,C 180,E1 -487.746,E2 -487.746} C_VEL
LIN {X 0,Y 608.442,Z 120.317,A -85,B 0,C 180,E1 -490.328,E2 -490.328} C_VEL
LIN {X 0,Y 608.477,Z 120.312,A -85,B 0,C 180,E1 -493.31,E2 -493.31} C_VEL
LIN {X 0,Y 608.464,Z 120.315,A -85,B 0,C 180,E1 -496.13,E2 -496.13} C_VEL
LIN {X 0,Y 608.453,Z 120.313,A -85,B 0,C 180,E1 -498.823,E2 -498.823} C_VEL
LIN {X 0,Y 608.457,Z 120.319,A -85,B 0,C 180,E1 -501.761,E2 -501.761} C_VEL
LIN {X 0,Y 608.441,Z 120.317,A -85,B 0,C 180,E1 -503.955,E2 -503.955} C_VEL
LIN {X 0,Y 608.443,Z 120.313,A -85,B 0,C 180,E1 -506.328,E2 -506.328} C_VEL
LIN {X 0,Y 608.449,Z 120.314,A -85,B 0,C 180,E1 -508.732,E2 -508.732} C_VEL
LIN {X 0,Y 608.47,Z 120.32,A -85,B 0,C 180,E1 -511.381,E2 -511.381} C_VEL
LIN {X 0,Y 608.432,Z 120.316,A -85,B 0,C 180,E1 -513.964,E2 -513.964} C_VEL
LIN {X 0,Y 608.451,Z 120.319,A -85,B 0,C 180,E1 -516.876,E2 -516.876} C_VEL
LIN {X 0,Y 608.455,Z 120.318,A -85,B 0,C 180,E1 -519.325,E2 -519.325} C_VEL
LIN {X 0,Y 608.43,Z 120.316,A -85,B 0,C 180,E1 -521.828,E2 -521.828} C_VEL
LIN {X 0,Y 608.473,Z 120.315,A -85,B 0,C 180,E1 -524.594,E2 -524.594} C_VEL
LIN {X 0,Y 608.456,Z 120.315,A -85,B 0,C 180,E1 -527.323,E2 -527.323} C_VEL
LIN {X 0,Y 608.454,Z 120.313,A -85,B 0,C 180,E1 -530.023,E2 -530.023} C_VEL
LIN {X 0,Y 608.462,Z 120.322,A -85,B 0,C 180,E1 -532.701,E2 -532.701} C_VEL
LIN {X 0,Y 608.467,Z 120.32,A -85,B 0,C 180,E1 -534.698,E2 -534.698} C_VEL
LIN {X 0,Y 608.447,Z 120.314,A -85,B 0,C 180,E1 -537.352,E2 -537.352} C_VEL
LIN {X 0,Y 608.477,Z 120.312,A -85,B 0,C 180,E1 -540,E2 -540} C_VEL
LIN {X 0,Y 608.468,Z 120.317,A -85,B 0,C 180,E1 -542.648,E2 -542.648} C_VEL
LIN {X 0,Y 608.434,Z 120.315,A -85,B 0,C 180,E1 -545.302,E2 -545.302} C_VEL
LIN {X 0,Y 608.478,Z 120.315,A -85,B 0,C 180,E1 -547.967,E2 -547.967} C_VEL
LIN {X 0,Y 608.441,Z 120.314,A -85,B 0,C 180,E1 -549.444,E2 -549.444} C_VEL
LIN {X 0,Y 607.78,Z 120.404,A -85,B 0,C 180,E1 -549.997,E2 -549.997} C_VEL
LIN {X 0,Y 604.939,Z 120.762,A -85,B 0,C 180,E1 -550.894,E2 -550.894} C_VEL
LIN {X 0,Y 602.531,Z 121.064,A -85,B 0,C 180,E1 -551.615,E2 -551.615} C_VEL
LIN {X 0,Y 601.488,Z 121.19,A -85,B 0,C 180,E1 -552.172,E2 -552.172} C_VEL
LIN {X 0,Y 601.399,Z 121.198,A -85,B 0,C 180,E1 -552.36,E2 -552.36} C_VEL
LIN {X 0,Y 601.39,Z 121.192,A -85,B 0,C 180,E1 -554.898,E2 -554.898} C_VEL
LIN {X 0,Y 601.379,Z 121.194,A -85,B 0,C 180,E1 -556.987,E2 -556.987} C_VEL
LIN {X 0,Y 601.394,Z 121.2,A -85,B 0,C 180,E1 -559.81,E2 -559.81} C_VEL
LIN {X 0,Y 601.401,Z 121.191,A -85,B 0,C 180,E1 -562.684,E2 -562.684} C_VEL
LIN {X 0,Y 601.384,Z 121.193,A -85,B 0,C 180,E1 -564.879,E2 -564.879} C_VEL
LIN {X 0,Y 601.404,Z 121.195,A -85,B 0,C 180,E1 -567.36,E2 -567.36} C_VEL
LIN {X 0,Y 601.4,Z 121.193,A -85,B 0,C 180,E1 -570.166,E2 -570.166} C_VEL
LIN {X 0,Y 601.394,Z 121.19,A -85,B 0,C 180,E1 -572.711,E2 -572.711} C_VEL
LIN {X 0,Y 601.379,Z 121.197,A -85,B 0,C 180,E1 -575.109,E2 -575.109} C_VEL
LIN {X 0,Y 601.432,Z 121.198,A -85,B 0,C 180,E1 -577.419,E2 -577.419} C_VEL
LIN {X 0,Y 601.378,Z 121.194,A -85,B 0,C 180,E1 -579.998,E2 -579.998} C_VEL
LIN {X 0,Y 601.374,Z 121.196,A -85,B 0,C 180,E1 -582.674,E2 -582.674} C_VEL
LIN {X 0,Y 601.4,Z 121.196,A -85,B 0,C 180,E1 -585.479,E2 -585.479} C_VEL
LIN {X 0,Y 601.404,Z 121.192,A -85,B 0,C 180,E1 -588.409,E2 -588.409} C_VEL
LIN {X 0,Y 601.393,Z 121.195,A -85,B 0,C 180,E1 -591.534,E2 -591.534} C_VEL
LIN {X 0,Y 601.371,Z 121.195,A -85,B 0,C 180,E1 -593.744,E2 -593.744} C_VEL
LIN {X 0,Y 601.409,Z 121.197,A -85,B 0,C 180,E1 -596.685,E2 -596.685} C_VEL
LIN {X 0,Y 601.392,Z 121.197,A -85,B 0,C 180,E1 -599.056,E2 -599.056} C_VEL
LIN {X 0,Y 601.387,Z 121.195,A -85,B 0,C 180,E1 -601.371,E2 -601.371} C_VEL
LIN {X 0,Y 601.37,Z 121.196,A -85,B 0,C 180,E1 -603.635,E2 -603.635} C_VEL
LIN {X 0,Y 601.418,Z 121.313,A -85,B 0,C 180,E1 -606.361,E2 -606.361} C_VEL
LIN {X 0,Y 601.719,Z 122.738,A -85,B 0,C 180,E1 -606.602,E2 -606.602} C_VEL
LIN {X 0,Y 601.664,Z 142.732,A -85,B 0,C 180,E1 -609.144,E2 -609.144} C_VEL
LIN {X 0,Y 601.622,Z 160.585,A -85,B 0,C 180,E1 -611.357,E2 -611.357} C_VEL
LIN {X 0,Y 602.03,Z 163.912,A -85,B 0,C 180,E1 -611.432,E2 -611.432} C_VEL
LIN {X 0,Y 601.885,Z 326.584,A -85,B 0,C 180,E1 -613.443,E2 -613.443} C_VEL
LIN {X 0,Y 601.849,Z 342.439,A -85,B 0,C 180,E1 -613.79,E2 -613.79} C_VEL
LIN {X 0,Y 601.767,Z 357.008,A -85,B 0,C 180,E1 -614.244,E2 -614.244} C_VEL
LIN {X 0,Y 601.704,Z 371.684,A -85,B 0,C 180,E1 -614.85,E2 -614.85} C_VEL
LIN {X 0,Y 601.658,Z 384.984,A -85,B 0,C 180,E1 -615.541,E2 -615.541} C_VEL
LIN {X 0,Y 601.604,Z 397.803,A -85,B 0,C 180,E1 -616.352,E2 -616.352} C_VEL
LIN {X 0,Y 601.541,Z 409.79,A -85,B 0,C 180,E1 -617.26,E2 -617.26} C_VEL
LIN {X 0,Y 601.489,Z 420.28,A -85,B 0,C 180,E1 -618.201,E2 -618.201} C_VEL
LIN {X 0,Y 601.43,Z 429.996,A -85,B 0,C 180,E1 -619.224,E2 -619.224} C_VEL
LIN {X 0,Y 601.428,Z 439.526,A -85,B 0,C 180,E1 -620.415,E2 -620.415} C_VEL
LIN {X 0,Y 601.378,Z 447.46,A -85,B 0,C 180,E1 -621.6,E2 -621.6} C_VEL
LIN {X 0,Y 601.368,Z 454.872,A -85,B 0,C 180,E1 -622.951,E2 -622.951} C_VEL
LIN {X 0,Y 601.373,Z 460.759,A -85,B 0,C 180,E1 -624.299,E2 -624.299} C_VEL
LIN {X 0,Y 601.327,Z 464.242,A -85,B 0,C 180,E1 -625.307,E2 -625.307} C_VEL
LIN {X 0,Y 601.336,Z 467.79,A -85,B 0,C 180,E1 -626.65,E2 -626.65} C_VEL
LIN {X 0,Y 601.343,Z 470.139,A -85,B 0,C 180,E1 -627.991,E2 -627.991} C_VEL
LIN {X 0,Y 601.334,Z 471.337,A -85,B 0,C 180,E1 -629.33,E2 -629.33} C_VEL
LIN {X 0,Y 601.335,Z 471.361,A -85,B 0,C 180,E1 -630.67,E2 -630.67} C_VEL
LIN {X 0,Y 601.343,Z 470.245,A -85,B 0,C 180,E1 -632.009,E2 -632.009} C_VEL
LIN {X 0,Y 601.339,Z 467.983,A -85,B 0,C 180,E1 -633.35,E2 -633.35} C_VEL
LIN {X 0,Y 601.328,Z 464.525,A -85,B 0,C 180,E1 -634.693,E2 -634.693} C_VEL
LIN {X 0,Y 601.358,Z 459.797,A -85,B 0,C 180,E1 -636.038,E2 -636.038} C_VEL
LIN {X 0,Y 601.366,Z 453.666,A -85,B 0,C 180,E1 -637.386,E2 -637.386} C_VEL
LIN {X 0,Y 601.389,Z 445.95,A -85,B 0,C 180,E1 -638.738,E2 -638.738} C_VEL
LIN {X 0,Y 601.428,Z 437.707,A -85,B 0,C 180,E1 -639.925,E2 -639.925} C_VEL
LIN {X 0,Y 601.443,Z 427.365,A -85,B 0,C 180,E1 -641.164,E2 -641.164} C_VEL
LIN {X 0,Y 601.501,Z 415.784,A -85,B 0,C 180,E1 -642.312,E2 -642.312} C_VEL
LIN {X 0,Y 601.557,Z 404.462,A -85,B 0,C 180,E1 -643.255,E2 -643.255} C_VEL
LIN {X 0,Y 601.624,Z 391.312,A -85,B 0,C 180,E1 -644.168,E2 -644.168} C_VEL
LIN {X 0,Y 601.657,Z 378.757,A -85,B 0,C 180,E1 -644.891,E2 -644.891} C_VEL
LIN {X 0,Y 601.74,Z 363.832,A -85,B 0,C 180,E1 -645.583,E2 -645.583} C_VEL
LIN {X 0,Y 601.819,Z 349.342,A -85,B 0,C 180,E1 -646.102,E2 -646.102} C_VEL
LIN {X 0,Y 601.859,Z 333.928,A -85,B 0,C 180,E1 -646.506,E2 -646.506} C_VEL
LIN {X 0,Y 601.9,Z 318.021,A -85,B 0,C 180,E1 -646.772,E2 -646.772} C_VEL
LIN {X 0,Y 601.928,Z 162.354,A -85,B 0,C 180,E1 -648.68,E2 -648.68} C_VEL
LIN {X 0,Y 601.602,Z 160.267,A -85,B 0,C 180,E1 -648.759,E2 -648.759} C_VEL
LIN {X 0,Y 601.685,Z 137.645,A -85,B 0,C 180,E1 -651.589,E2 -651.589} C_VEL
LIN {X 0,Y 601.744,Z 123.439,A -85,B 0,C 180,E1 -653.397,E2 -653.397} C_VEL
LIN {X 0,Y 601.421,Z 121.309,A -85,B 0,C 180,E1 -653.73,E2 -653.73} C_VEL
LIN {X 0,Y 601.363,Z 121.196,A -85,B 0,C 180,E1 -656.366,E2 -656.366} C_VEL
LIN {X 0,Y 601.387,Z 121.196,A -85,B 0,C 180,E1 -658.78,E2 -658.78} C_VEL
LIN {X 0,Y 601.376,Z 121.197,A -85,B 0,C 180,E1 -661.729,E2 -661.729} C_VEL
LIN {X 0,Y 601.395,Z 121.192,A -85,B 0,C 180,E1 -664.121,E2 -664.121} C_VEL
LIN {X 0,Y 601.429,Z 121.192,A -85,B 0,C 180,E1 -667.42,E2 -667.42} C_VEL
LIN {X 0,Y 601.375,Z 121.194,A -85,B 0,C 180,E1 -669.998,E2 -669.998} C_VEL
LIN {X 0,Y 601.374,Z 121.201,A -85,B 0,C 180,E1 -672.674,E2 -672.674} C_VEL
LIN {X 0,Y 601.4,Z 121.192,A -85,B 0,C 180,E1 -675.479,E2 -675.479} C_VEL
LIN {X 0,Y 601.408,Z 121.195,A -85,B 0,C 180,E1 -678.409,E2 -678.409} C_VEL
LIN {X 0,Y 601.397,Z 121.198,A -85,B 0,C 180,E1 -680.872,E2 -680.872} C_VEL
LIN {X 0,Y 601.387,Z 121.193,A -85,B 0,C 180,E1 -683.416,E2 -683.416} C_VEL
LIN {X 0,Y 601.412,Z 121.193,A -85,B 0,C 180,E1 -686.068,E2 -686.068} C_VEL
LIN {X 0,Y 601.392,Z 121.193,A -85,B 0,C 180,E1 -689.056,E2 -689.056} C_VEL
LIN {X 0,Y 601.391,Z 121.192,A -85,B 0,C 180,E1 -691.371,E2 -691.371} C_VEL
LIN {X 0,Y 601.41,Z 121.198,A -85,B 0,C 180,E1 -694.134,E2 -694.134} C_VEL
LIN {X 0,Y 601.383,Z 121.198,A -85,B 0,C 180,E1 -696.588,E2 -696.588} C_VEL
LIN {X 0,Y 601.401,Z 121.192,A -85,B 0,C 180,E1 -699.477,E2 -699.477} C_VEL
LIN {X 0,Y 601.386,Z 121.199,A -85,B 0,C 180,E1 -702.311,E2 -702.311} C_VEL
LIN {X 0,Y 601.399,Z 121.195,A -85,B 0,C 180,E1 -704.408,E2 -704.408} C_VEL
LIN {X 0,Y 601.403,Z 121.193,A -85,B 0,C 180,E1 -706.484,E2 -706.484} C_VEL
LIN {X 0,Y 601.376,Z 121.196,A -85,B 0,C 180,E1 -709.223,E2 -709.223} C_VEL
LIN {X 0,Y 601.438,Z 121.194,A -85,B 0,C 180,E1 -711.939,E2 -711.939} C_VEL
LIN {X 0,Y 601.403,Z 121.191,A -85,B 0,C 180,E1 -714.636,E2 -714.636} C_VEL
LIN {X 0,Y 601.428,Z 121.193,A -85,B 0,C 180,E1 -717.321,E2 -717.321} C_VEL
LIN {X 0,Y 601.446,Z 121.189,A -85,B 0,C 180,E1 -720,E2 -720} C_VEL
LIN {X 0,Y 601.413,Z 121.19,A -85,B 0,C 180,E1 -722.679,E2 -722.679} C_VEL
LIN {X 0,Y 601.429,Z 121.197,A -85,B 0,C 180,E1 -725.364,E2 -725.364} C_VEL
LIN {X 0,Y 601.434,Z 121.187,A -85,B 0,C 180,E1 -728.061,E2 -728.061} C_VEL
LIN {X 0,Y 601.413,Z 121.196,A -85,B 0,C 180,E1 -731.005,E2 -731.005} C_VEL
LIN {X 0,Y 601.418,Z 121.193,A -85,B 0,C 180,E1 -733.516,E2 -733.516} C_VEL
LIN {X 0,Y 601.421,Z 121.189,A -85,B 0,C 180,E1 -736.287,E2 -736.287} C_VEL
LIN {X 0,Y 601.415,Z 121.198,A -85,B 0,C 180,E1 -739.099,E2 -739.099} C_VEL
LIN {X 0,Y 601.405,Z 121.195,A -85,B 0,C 180,E1 -741.239,E2 -741.239} C_VEL
LIN {X 0,Y 601.412,Z 121.191,A -85,B 0,C 180,E1 -744.142,E2 -744.142} C_VEL
LIN {X 0,Y 601.454,Z 121.189,A -85,B 0,C 180,E1 -747.111,E2 -747.111} C_VEL
LIN {X 0,Y 601.411,Z 121.191,A -85,B 0,C 180,E1 -749.393,E2 -749.393} C_VEL
LIN {X 0,Y 601.396,Z 121.191,A -85,B 0,C 180,E1 -751.727,E2 -751.727} C_VEL
LIN {X 0,Y 601.42,Z 121.19,A -85,B 0,C 180,E1 -754.119,E2 -754.119} C_VEL
LIN {X 0,Y 601.437,Z 121.187,A -85,B 0,C 180,E1 -757.382,E2 -757.382} C_VEL
LIN {X 0,Y 601.401,Z 121.194,A -85,B 0,C 180,E1 -759.996,E2 -759.996} C_VEL
LIN {X 0,Y 601.416,Z 121.194,A -85,B 0,C 180,E1 -762.67,E2 -762.67} C_VEL
LIN {X 0,Y 601.399,Z 121.192,A -85,B 0,C 180,E1 -765.479,E2 -765.479} C_VEL
LIN {X 0,Y 601.424,Z 121.194,A -85,B 0,C 180,E1 -768.407,E2 -768.407} C_VEL
LIN {X 0,Y 601.438,Z 121.187,A -85,B 0,C 180,E1 -770.875,E2 -770.875} C_VEL
LIN {X 0,Y 601.4,Z 121.193,A -85,B 0,C 180,E1 -773.417,E2 -773.417} C_VEL
LIN {X 0,Y 601.434,Z 121.195,A -85,B 0,C 180,E1 -776.064,E2 -776.064} C_VEL
LIN {X 0,Y 601.42,Z 121.189,A -85,B 0,C 180,E1 -778.545,E2 -778.545} C_VEL
LIN {X 0,Y 601.425,Z 121.192,A -85,B 0,C 180,E1 -781.373,E2 -781.373} C_VEL
LIN {X 0,Y 601.401,Z 121.201,A -85,B 0,C 180,E1 -783.636,E2 -783.636} C_VEL
LIN {X 0,Y 601.459,Z 121.361,A -85,B 0,C 180,E1 -785.4,E2 -785.4} C_VEL
LIN {X 0,Y 601.816,Z 124.966,A -85,B 0,C 180,E1 -785.875,E2 -785.875} C_VEL
LIN {X 0,Y 601.694,Z 147.322,A -85,B 0,C 180,E1 -788.592,E2 -788.592} C_VEL
LIN {X 0,Y 601.61,Z 169.946,A -85,B 0,C 180,E1 -791.287,E2 -791.287} C_VEL
LIN {X 0,Y 602.044,Z 172.386,A -85,B 0,C 180,E1 -791.369,E2 -791.369} C_VEL
LIN {X 0,Y 601.9,Z 336.06,A -85,B 0,C 180,E1 -793.389,E2 -793.389} C_VEL
LIN {X 0,Y 601.835,Z 351.707,A -85,B 0,C 180,E1 -793.724,E2 -793.724} C_VEL
LIN {X 0,Y 601.781,Z 367.045,A -85,B 0,C 180,E1 -794.201,E2 -794.201} C_VEL
LIN {X 0,Y 601.722,Z 380.759,A -85,B 0,C 180,E1 -794.764,E2 -794.764} C_VEL
LIN {X 0,Y 601.66,Z 394.233,A -85,B 0,C 180,E1 -795.455,E2 -795.455} C_VEL
LIN {X 0,Y 601.617,Z 407.449,A -85,B 0,C 180,E1 -796.283,E2 -796.283} C_VEL
LIN {X 0,Y 601.531,Z 419.284,A -85,B 0,C 180,E1 -797.174,E2 -797.174} C_VEL
LIN {X 0,Y 601.488,Z 430.747,A -85,B 0,C 180,E1 -798.201,E2 -798.201} C_VEL
LIN {X 0,Y 601.43,Z 440.388,A -85,B 0,C 180,E1 -799.224,E2 -799.224} C_VEL
LIN {X 0,Y 601.428,Z 449.854,A -85,B 0,C 180,E1 -800.414,E2 -800.414} C_VEL
LIN {X 0,Y 601.369,Z 457.73,A -85,B 0,C 180,E1 -801.6,E2 -801.6} C_VEL
LIN {X 0,Y 601.367,Z 465.088,A -85,B 0,C 180,E1 -802.951,E2 -802.951} C_VEL
LIN {X 0,Y 601.373,Z 470.924,A -85,B 0,C 180,E1 -804.299,E2 -804.299} C_VEL
LIN {X 0,Y 601.33,Z 474.383,A -85,B 0,C 180,E1 -805.307,E2 -805.307} C_VEL
LIN {X 0,Y 601.337,Z 477.886,A -85,B 0,C 180,E1 -806.65,E2 -806.65} C_VEL
LIN {X 0,Y 601.343,Z 480.192,A -85,B 0,C 180,E1 -807.991,E2 -807.991} C_VEL
LIN {X 0,Y 601.335,Z 481.35,A -85,B 0,C 180,E1 -809.33,E2 -809.33} C_VEL
LIN {X 0,Y 601.335,Z 481.35,A -85,B 0,C 180,E1 -810.67,E2 -810.67} C_VEL
LIN {X 0,Y 601.343,Z 480.192,A -85,B 0,C 180,E1 -812.009,E2 -812.009} C_VEL
LIN {X 0,Y 601.337,Z 477.886,A -85,B 0,C 180,E1 -813.35,E2 -813.35} C_VEL
LIN {X 0,Y 601.329,Z 474.383,A -85,B 0,C 180,E1 -814.693,E2 -814.693} C_VEL
LIN {X 0,Y 601.357,Z 469.608,A -85,B 0,C 180,E1 -816.038,E2 -816.038} C_VEL
LIN {X 0,Y 601.365,Z 463.425,A -85,B 0,C 180,E1 -817.386,E2 -817.386} C_VEL
LIN {X 0,Y 601.388,Z 455.653,A -85,B 0,C 180,E1 -818.738,E2 -818.738} C_VEL
LIN {X 0,Y 601.427,Z 447.37,A -85,B 0,C 180,E1 -819.925,E2 -819.925} C_VEL
LIN {X 0,Y 601.46,Z 436.932,A -85,B 0,C 180,E1 -821.165,E2 -821.165} C_VEL
LIN {X 0,Y 601.514,Z 427.192,A -85,B 0,C 180,E1 -822.14,E2 -822.14} C_VEL
LIN {X 0,Y 601.57,Z 415.016,A -85,B 0,C 180,E1 -823.168,E2 -823.168} C_VEL
LIN {X 0,Y 601.606,Z 403.076,A -85,B 0,C 180,E1 -824.012,E2 -824.012} C_VEL
LIN {X 0,Y 601.665,Z 389.525,A -85,B 0,C 180,E1 -824.804,E2 -824.804} C_VEL
LIN {X 0,Y 601.742,Z 374.84,A -85,B 0,C 180,E1 -825.496,E2 -825.496} C_VEL
LIN {X 0,Y 601.794,Z 360.617,A -85,B 0,C 180,E1 -826.016,E2 -826.016} C_VEL
LIN {X 0,Y 601.865,Z 345.581,A -85,B 0,C 180,E1 -826.422,E2 -826.422} C_VEL
LIN {X 0,Y 601.901,Z 330.484,A -85,B 0,C 180,E1 -826.692,E2 -826.692} C_VEL
LIN {X 0,Y 601.995,Z 172.25,A -85,B 0,C 180,E1 -828.635,E2 -828.635} C_VEL
LIN {X 0,Y 601.619,Z 170.1,A -85,B 0,C 180,E1 -828.7,E2 -828.7} C_VEL
LIN {X 0,Y 601.688,Z 148.812,A -85,B 0,C 180,E1 -831.229,E2 -831.229} C_VEL
LIN {X 0,Y 601.818,Z 126.457,A -85,B 0,C 180,E1 -833.942,E2 -833.942} C_VEL
LIN {X 0,Y 601.772,Z 123.046,A -85,B 0,C 180,E1 -834.363,E2 -834.363} C_VEL
LIN {X 0,Y 601.443,Z 121.244,A -85,B 0,C 180,E1 -834.64,E2 -834.64} C_VEL
LIN {X 0,Y 601.413,Z 121.19,A -85,B 0,C 180,E1 -837.362,E2 -837.362} C_VEL
LIN {X 0,Y 601.429,Z 121.198,A -85,B 0,C 180,E1 -840.164,E2 -840.164} C_VEL
LIN {X 0,Y 601.417,Z 121.19,A -85,B 0,C 180,E1 -842.715,E2 -842.715} C_VEL
LIN {X 0,Y 601.389,Z 121.193,A -85,B 0,C 180,E1 -845.111,E2 -845.111} C_VEL
LIN {X 0,Y 601.437,Z 121.189,A -85,B 0,C 180,E1 -847.419,E2 -847.419} C_VEL
LIN {X 0,Y 601.412,Z 121.199,A -85,B 0,C 180,E1 -849.995,E2 -849.995} C_VEL
LIN {X 0,Y 601.408,Z 121.19,A -85,B 0,C 180,E1 -852.671,E2 -852.671} C_VEL
LIN {X 0,Y 601.427,Z 121.193,A -85,B 0,C 180,E1 -855.482,E2 -855.482} C_VEL
LIN {X 0,Y 601.42,Z 121.189,A -85,B 0,C 180,E1 -858.408,E2 -858.408} C_VEL
LIN {X 0,Y 601.429,Z 121.197,A -85,B 0,C 180,E1 -861.53,E2 -861.53} C_VEL
LIN {X 0,Y 601.382,Z 121.194,A -85,B 0,C 180,E1 -864.245,E2 -864.245} C_VEL
LIN {X 0,Y 601.417,Z 121.188,A -85,B 0,C 180,E1 -866.686,E2 -866.686} C_VEL
LIN {X 0,Y 601.413,Z 121.194,A -85,B 0,C 180,E1 -869.058,E2 -869.058} C_VEL
LIN {X 0,Y 601.43,Z 121.197,A -85,B 0,C 180,E1 -871.373,E2 -871.373} C_VEL
LIN {X 0,Y 601.395,Z 121.195,A -85,B 0,C 180,E1 -873.636,E2 -873.636} C_VEL
LIN {X 0,Y 601.438,Z 121.188,A -85,B 0,C 180,E1 -875.859,E2 -875.859} C_VEL
LIN {X 0,Y 601.407,Z 121.195,A -85,B 0,C 180,E1 -878.761,E2 -878.761} C_VEL
LIN {X 0,Y 601.391,Z 121.194,A -85,B 0,C 180,E1 -881.607,E2 -881.607} C_VEL
LIN {X 0,Y 601.412,Z 121.192,A -85,B 0,C 180,E1 -884.409,E2 -884.409} C_VEL
LIN {X 0,Y 601.407,Z 121.196,A -85,B 0,C 180,E1 -887.172,E2 -887.172} C_VEL
LIN {X 0,Y 601.428,Z 121.187,A -85,B 0,C 180,E1 -889.905,E2 -889.905} C_VEL
LIN {X 0,Y 601.44,Z 121.195,A -85,B 0,C 180,E1 -892.615,E2 -892.615} C_VEL
LIN {X 0,Y 601.397,Z 121.192,A -85,B 0,C 180,E1 -895.308,E2 -895.308} C_VEL
LIN {X 0,Y 601.436,Z 121.188,A -85,B 0,C 180,E1 -897.991,E2 -897.991} C_VEL
LIN {X 0,Y 601.444,Z 121.192,A -85,B 0,C 180,E1 -900.67,E2 -900.67} C_VEL
LIN {X 0,Y 601.376,Z 121.194,A -85,B 0,C 180,E1 -903.35,E2 -903.35} C_VEL
LIN {X 0,Y 601.438,Z 121.192,A -85,B 0,C 180,E1 -906.037,E2 -906.037} C_VEL
LIN {X 0,Y 601.399,Z 121.194,A -85,B 0,C 180,E1 -908.738,E2 -908.738} C_VEL
LIN {X 0,Y 601.407,Z 121.191,A -85,B 0,C 180,E1 -911.459,E2 -911.459} C_VEL
LIN {X 0,Y 601.399,Z 121.198,A -85,B 0,C 180,E1 -912.36,E2 -912.36} C_VEL
LIN {X 0,Y 600.719,Z 121.278,A -85,B 0,C 180,E1 -912.92,E2 -912.92} C_VEL
LIN {X 0,Y 597.859,Z 121.638,A -85,B 0,C 180,E1 -913.828,E2 -913.828} C_VEL
LIN {X 0,Y 595.452,Z 121.934,A -85,B 0,C 180,E1 -914.558,E2 -914.558} C_VEL
LIN {X 0,Y 594.42,Z 122.06,A -85,B 0,C 180,E1 -915.121,E2 -915.121} C_VEL
LIN {X 0,Y 594.337,Z 122.071,A -85,B 0,C 180,E1 -915.312,E2 -915.312} C_VEL
LIN {X 0,Y 594.337,Z 122.08,A -85,B 0,C 180,E1 -917.906,E2 -917.906} C_VEL
LIN {X 0,Y 594.381,Z 122.065,A -85,B 0,C 180,E1 -920.776,E2 -920.776} C_VEL
LIN {X 0,Y 594.357,Z 122.077,A -85,B 0,C 180,E1 -923.706,E2 -923.706} C_VEL
LIN {X 0,Y 594.361,Z 122.074,A -85,B 0,C 180,E1 -926.017,E2 -926.017} C_VEL
LIN {X 0,Y 594.352,Z 122.072,A -85,B 0,C 180,E1 -928.228,E2 -928.228} C_VEL
LIN {X 0,Y 594.363,Z 122.066,A -85,B 0,C 180,E1 -930.561,E2 -930.561} C_VEL
LIN {X 0,Y 594.372,Z 122.065,A -85,B 0,C 180,E1 -932.951,E2 -932.951} C_VEL
LIN {X 0,Y 594.324,Z 122.081,A -85,B 0,C 180,E1 -935.411,E2 -935.411} C_VEL
LIN {X 0,Y 594.366,Z 122.069,A -85,B 0,C 180,E1 -937.942,E2 -937.942} C_VEL
LIN {X 0,Y 594.363,Z 122.068,A -85,B 0,C 180,E1 -940.82,E2 -940.82} C_VEL
LIN {X 0,Y 594.344,Z 122.072,A -85,B 0,C 180,E1 -943.837,E2 -943.837} C_VEL
LIN {X 0,Y 594.343,Z 122.072,A -85,B 0,C 180,E1 -946.698,E2 -946.698} C_VEL
LIN {X 0,Y 594.359,Z 122.072,A -85,B 0,C 180,E1 -949.432,E2 -949.432} C_VEL
LIN {X 0,Y 594.38,Z 122.067,A -85,B 0,C 180,E1 -952.393,E2 -952.393} C_VEL
LIN {X 0,Y 594.36,Z 122.071,A -85,B 0,C 180,E1 -955.419,E2 -955.419} C_VEL
LIN {X 0,Y 594.337,Z 122.072,A -85,B 0,C 180,E1 -957.851,E2 -957.851} C_VEL
LIN {X 0,Y 594.333,Z 122.071,A -85,B 0,C 180,E1 -960.221,E2 -960.221} C_VEL
LIN {X 0,Y 594.356,Z 122.072,A -85,B 0,C 180,E1 -963.299,E2 -963.299} C_VEL
LIN {X 0,Y 594.406,Z 122.254,A -85,B 0,C 180,E1 -966.204,E2 -966.204} C_VEL
LIN {X 0,Y 594.88,Z 125.582,A -85,B 0,C 180,E1 -966.686,E2 -966.686} C_VEL
LIN {X 0,Y 594.752,Z 146.877,A -85,B 0,C 180,E1 -969.418,E2 -969.418} C_VEL
LIN {X 0,Y 594.676,Z 160.605,A -85,B 0,C 180,E1 -971.132,E2 -971.132} C_VEL
LIN {X 0,Y 595.317,Z 165.208,A -85,B 0,C 180,E1 -971.231,E2 -971.231} C_VEL
LIN {X 0,Y 595.097,Z 325.872,A -85,B 0,C 180,E1 -973.236,E2 -973.236} C_VEL
LIN {X 0,Y 595.03,Z 341.682,A -85,B 0,C 180,E1 -973.577,E2 -973.577} C_VEL
LIN {X 0,Y 594.924,Z 357.022,A -85,B 0,C 180,E1 -974.058,E2 -974.058} C_VEL
LIN {X 0,Y 594.818,Z 371.694,A -85,B 0,C 180,E1 -974.671,E2 -974.671} C_VEL
LIN {X 0,Y 594.744,Z 384.997,A -85,B 0,C 180,E1 -975.369,E2 -975.369} C_VEL
LIN {X 0,Y 594.67,Z 397.991,A -85,B 0,C 180,E1 -976.201,E2 -976.201} C_VEL
LIN {X 0,Y 594.552,Z 410.858,A -85,B 0,C 180,E1 -977.195,E2 -977.195} C_VEL
LIN {X 0,Y 594.468,Z 422.062,A -85,B 0,C 180,E1 -978.233,E2 -978.233} C_VEL
LIN {X 0,Y 594.412,Z 432.946,A -85,B 0,C 180,E1 -979.44,E2 -979.44} C_VEL
LIN {X 0,Y 594.356,Z 441.991,A -85,B 0,C 180,E1 -980.643,E2 -980.643} C_VEL
LIN {X 0,Y 594.324,Z 449.485,A -85,B 0,C 180,E1 -981.842,E2 -981.842} C_VEL
LIN {X 0,Y 594.277,Z 456.49,A -85,B 0,C 180,E1 -983.208,E2 -983.208} C_VEL
LIN {X 0,Y 594.273,Z 461.999,A -85,B 0,C 180,E1 -984.571,E2 -984.571} C_VEL
LIN {X 0,Y 594.253,Z 466.171,A -85,B 0,C 180,E1 -985.931,E2 -985.931} C_VEL
LIN {X 0,Y 594.221,Z 469.112,A -85,B 0,C 180,E1 -987.288,E2 -987.288} C_VEL
LIN {X 0,Y 594.243,Z 470.88,A -85,B 0,C 180,E1 -988.645,E2 -988.645} C_VEL
LIN {X 0,Y 594.234,Z 471.496,A -85,B 0,C 180,E1 -990,E2 -990} C_VEL
LIN {X 0,Y 594.245,Z 470.944,A -85,B 0,C 180,E1 -991.355,E2 -991.355} C_VEL
LIN {X 0,Y 594.224,Z 469.259,A -85,B 0,C 180,E1 -992.712,E2 -992.712} C_VEL
LIN {X 0,Y 594.253,Z 466.406,A -85,B 0,C 180,E1 -994.069,E2 -994.069} C_VEL
LIN {X 0,Y 594.273,Z 462.325,A -85,B 0,C 180,E1 -995.429,E2 -995.429} C_VEL
LIN {X 0,Y 594.277,Z 456.915,A -85,B 0,C 180,E1 -996.792,E2 -996.792} C_VEL
LIN {X 0,Y 594.323,Z 450.016,A -85,B 0,C 180,E1 -998.158,E2 -998.158} C_VEL
LIN {X 0,Y 594.339,Z 441.413,A -85,B 0,C 180,E1 -999.529,E2 -999.529} C_VEL
LIN {X 0,Y 594.401,Z 432.263,A -85,B 0,C 180,E1 -1000.732,E2 -1000.732} C_VEL
LIN {X 0,Y 594.466,Z 421.21,A -85,B 0,C 180,E1 -1001.94,E2 -1001.94} C_VEL
LIN {X 0,Y 594.56,Z 409.835,A -85,B 0,C 180,E1 -1002.979,E2 -1002.979} C_VEL
LIN {X 0,Y 594.66,Z 397.451,A -85,B 0,C 180,E1 -1003.925,E2 -1003.925} C_VEL
LIN {X 0,Y 594.723,Z 385.042,A -85,B 0,C 180,E1 -1004.719,E2 -1004.719} C_VEL
LIN {X 0,Y 594.852,Z 371.742,A -85,B 0,C 180,E1 -1005.416,E2 -1005.416} C_VEL
LIN {X 0,Y 594.921,Z 357.069,A -85,B 0,C 180,E1 -1006.03,E2 -1006.03} C_VEL
LIN {X 0,Y 595.036,Z 341.909,A -85,B 0,C 180,E1 -1006.507,E2 -1006.507} C_VEL
LIN {X 0,Y 595.087,Z 326.762,A -85,B 0,C 180,E1 -1006.839,E2 -1006.839} C_VEL
LIN {X 0,Y 595.189,Z 237.122,A -85,B 0,C 180,E1 -1007.968,E2 -1007.968} C_VEL
LIN {X 0,Y 595.245,Z 163.44,A -85,B 0,C 180,E1 -1008.884,E2 -1008.884} C_VEL
LIN {X 0,Y 594.685,Z 160.647,A -85,B 0,C 180,E1 -1008.955,E2 -1008.955} C_VEL
LIN {X 0,Y 594.778,Z 140.481,A -85,B 0,C 180,E1 -1011.488,E2 -1011.488} C_VEL
LIN {X 0,Y 594.871,Z 124.855,A -85,B 0,C 180,E1 -1013.499,E2 -1013.499} C_VEL
LIN {X 0,Y 594.383,Z 122.246,A -85,B 0,C 180,E1 -1013.89,E2 -1013.89} C_VEL
LIN {X 0,Y 594.348,Z 122.072,A -85,B 0,C 180,E1 -1016.701,E2 -1016.701} C_VEL
LIN {X 0,Y 594.33,Z 122.072,A -85,B 0,C 180,E1 -1019.779,E2 -1019.779} C_VEL
LIN {X 0,Y 594.332,Z 122.072,A -85,B 0,C 180,E1 -1022.149,E2 -1022.149} C_VEL
LIN {X 0,Y 594.355,Z 122.071,A -85,B 0,C 180,E1 -1024.582,E2 -1024.582} C_VEL
LIN {X 0,Y 594.375,Z 122.069,A -85,B 0,C 180,E1 -1027.606,E2 -1027.606} C_VEL
LIN {X 0,Y 594.339,Z 122.074,A -85,B 0,C 180,E1 -1030.57,E2 -1030.57} C_VEL
LIN {X 0,Y 594.342,Z 122.073,A -85,B 0,C 180,E1 -1033.302,E2 -1033.302} C_VEL
LIN {X 0,Y 594.344,Z 122.072,A -85,B 0,C 180,E1 -1036.163,E2 -1036.163} C_VEL
LIN {X 0,Y 594.36,Z 122.069,A -85,B 0,C 180,E1 -1039.18,E2 -1039.18} C_VEL
LIN {X 0,Y 594.35,Z 122.071,A -85,B 0,C 180,E1 -1042.056,E2 -1042.056} C_VEL
LIN {X 0,Y 594.321,Z 122.081,A -85,B 0,C 180,E1 -1044.681,E2 -1044.681} C_VEL
LIN {X 0,Y 594.37,Z 122.066,A -85,B 0,C 180,E1 -1047.09,E2 -1047.09} C_VEL
LIN {X 0,Y 594.365,Z 122.067,A -85,B 0,C 180,E1 -1049.676,E2 -1049.676} C_VEL
LIN {X 0,Y 594.36,Z 122.075,A -85,B 0,C 180,E1 -1052.538,E2 -1052.538} C_VEL
LIN {X 0,Y 594.361,Z 122.07,A -85,B 0,C 180,E1 -1054.806,E2 -1054.806} C_VEL
LIN {X 0,Y 594.345,Z 122.074,A -85,B 0,C 180,E1 -1057.766,E2 -1057.766} C_VEL
LIN {X 0,Y 594.357,Z 122.075,A -85,B 0,C 180,E1 -1059.946,E2 -1059.946} C_VEL
LIN {X 0,Y 594.331,Z 122.072,A -85,B 0,C 180,E1 -1062.805,E2 -1062.805} C_VEL
LIN {X 0,Y 594.389,Z 122.072,A -85,B 0,C 180,E1 -1065.828,E2 -1065.828} C_VEL
LIN {X 0,Y 594.376,Z 122.069,A -85,B 0,C 180,E1 -1068.404,E2 -1068.404} C_VEL
LIN {X 0,Y 594.364,Z 122.068,A -85,B 0,C 180,E1 -1071.158,E2 -1071.158} C_VEL
LIN {X 0,Y 594.384,Z 122.073,A -85,B 0,C 180,E1 -1073.891,E2 -1073.891} C_VEL
LIN {X 0,Y 594.329,Z 122.071,A -85,B 0,C 180,E1 -1076.61,E2 -1076.61} C_VEL
LIN {X 0,Y 594.349,Z 122.069,A -85,B 0,C 180,E1 -1078.645,E2 -1078.645} C_VEL
LIN {X 0,Y 594.397,Z 122.064,A -85,B 0,C 180,E1 -1080.677,E2 -1080.677} C_VEL
LIN {X 0,Y 594.374,Z 122.075,A -85,B 0,C 180,E1 -1083.389,E2 -1083.389} C_VEL
LIN {X 0,Y 594.381,Z 122.066,A -85,B 0,C 180,E1 -1086.109,E2 -1086.109} C_VEL
LIN {X 0,Y 594.369,Z 122.07,A -85,B 0,C 180,E1 -1088.842,E2 -1088.842} C_VEL
LIN {X 0,Y 594.395,Z 122.068,A -85,B 0,C 180,E1 -1091.596,E2 -1091.596} C_VEL
LIN {X 0,Y 594.381,Z 122.066,A -85,B 0,C 180,E1 -1094.377,E2 -1094.377} C_VEL
LIN {X 0,Y 594.377,Z 122.074,A -85,B 0,C 180,E1 -1097.194,E2 -1097.194} C_VEL
LIN {X 0,Y 594.365,Z 122.067,A -85,B 0,C 180,E1 -1100.054,E2 -1100.054} C_VEL
LIN {X 0,Y 594.355,Z 122.078,A -85,B 0,C 180,E1 -1102.968,E2 -1102.968} C_VEL
LIN {X 0,Y 594.373,Z 122.07,A -85,B 0,C 180,E1 -1105.193,E2 -1105.193} C_VEL
LIN {X 0,Y 594.37,Z 122.068,A -85,B 0,C 180,E1 -1107.523,E2 -1107.523} C_VEL
LIN {X 0,Y 594.369,Z 122.071,A -85,B 0,C 180,E1 -1110.325,E2 -1110.325} C_VEL
LIN {X 0,Y 594.378,Z 122.068,A -85,B 0,C 180,E1 -1112.95,E2 -1112.95} C_VEL
LIN {X 0,Y 594.35,Z 122.069,A -85,B 0,C 180,E1 -1115.409,E2 -1115.409} C_VEL
LIN {X 0,Y 594.382,Z 122.068,A -85,B 0,C 180,E1 -1117.941,E2 -1117.941} C_VEL
LIN {X 0,Y 594.376,Z 122.068,A -85,B 0,C 180,E1 -1120.822,E2 -1120.822} C_VEL
LIN {X 0,Y 594.368,Z 122.067,A -85,B 0,C 180,E1 -1123.299,E2 -1123.299} C_VEL
LIN {X 0,Y 594.362,Z 122.076,A -85,B 0,C 180,E1 -1126.161,E2 -1126.161} C_VEL
LIN {X 0,Y 594.381,Z 122.07,A -85,B 0,C 180,E1 -1128.536,E2 -1128.536} C_VEL
LIN {X 0,Y 594.387,Z 122.065,A -85,B 0,C 180,E1 -1131.295,E2 -1131.295} C_VEL
LIN {X 0,Y 594.352,Z 122.076,A -85,B 0,C 180,E1 -1133.755,E2 -1133.755} C_VEL
LIN {X 0,Y 594.38,Z 122.07,A -85,B 0,C 180,E1 -1136.239,E2 -1136.239} C_VEL
LIN {X 0,Y 594.37,Z 122.066,A -85,B 0,C 180,E1 -1138.65,E2 -1138.65} C_VEL
LIN {X 0,Y 594.382,Z 122.067,A -85,B 0,C 180,E1 -1141.042,E2 -1141.042} C_VEL
LIN {X 0,Y 594.387,Z 122.072,A -85,B 0,C 180,E1 -1143.977,E2 -1143.977} C_VEL
LIN {X 0,Y 594.409,Z 122.284,A -85,B 0,C 180,E1 -1145.208,E2 -1145.208} C_VEL
LIN {X 0,Y 594.974,Z 126.456,A -85,B 0,C 180,E1 -1145.765,E2 -1145.765} C_VEL
LIN {X 0,Y 594.84,Z 147.322,A -85,B 0,C 180,E1 -1148.333,E2 -1148.333} C_VEL
LIN {X 0,Y 594.712,Z 170.226,A -85,B 0,C 180,E1 -1151.083,E2 -1151.083} C_VEL
LIN {X 0,Y 595.329,Z 173.772,A -85,B 0,C 180,E1 -1151.168,E2 -1151.168} C_VEL
LIN {X 0,Y 595.102,Z 335.958,A -85,B 0,C 180,E1 -1153.192,E2 -1153.192} C_VEL
LIN {X 0,Y 595.027,Z 351.706,A -85,B 0,C 180,E1 -1153.533,E2 -1153.533} C_VEL
LIN {X 0,Y 594.945,Z 367.043,A -85,B 0,C 180,E1 -1154.015,E2 -1154.015} C_VEL
LIN {X 0,Y 594.851,Z 380.762,A -85,B 0,C 180,E1 -1154.584,E2 -1154.584} C_VEL
LIN {X 0,Y 594.735,Z 394.236,A -85,B 0,C 180,E1 -1155.282,E2 -1155.282} C_VEL
LIN {X 0,Y 594.681,Z 406.792,A -85,B 0,C 180,E1 -1156.075,E2 -1156.075} C_VEL
LIN {X 0,Y 594.56,Z 419.286,A -85,B 0,C 180,E1 -1157.021,E2 -1157.021} C_VEL
LIN {X 0,Y 594.465,Z 430.748,A -85,B 0,C 180,E1 -1158.06,E2 -1158.06} C_VEL
LIN {X 0,Y 594.388,Z 440.389,A -85,B 0,C 180,E1 -1159.095,E2 -1159.095} C_VEL
LIN {X 0,Y 594.366,Z 449.855,A -85,B 0,C 180,E1 -1160.3,E2 -1160.3} C_VEL
LIN {X 0,Y 594.312,Z 457.731,A -85,B 0,C 180,E1 -1161.499,E2 -1161.499} C_VEL
LIN {X 0,Y 594.291,Z 465.088,A -85,B 0,C 180,E1 -1162.867,E2 -1162.867} C_VEL
LIN {X 0,Y 594.299,Z 470.924,A -85,B 0,C 180,E1 -1164.231,E2 -1164.231} C_VEL
LIN {X 0,Y 594.232,Z 474.384,A -85,B 0,C 180,E1 -1165.251,E2 -1165.251} C_VEL
LIN {X 0,Y 594.257,Z 477.887,A -85,B 0,C 180,E1 -1166.61,E2 -1166.61} C_VEL
LIN {X 0,Y 594.241,Z 480.193,A -85,B 0,C 180,E1 -1167.967,E2 -1167.967} C_VEL
LIN {X 0,Y 594.235,Z 481.35,A -85,B 0,C 180,E1 -1169.322,E2 -1169.322} C_VEL
LIN {X 0,Y 594.235,Z 481.35,A -85,B 0,C 180,E1 -1170.678,E2 -1170.678} C_VEL
LIN {X 0,Y 594.241,Z 480.192,A -85,B 0,C 180,E1 -1172.033,E2 -1172.033} C_VEL
LIN {X 0,Y 594.257,Z 477.886,A -85,B 0,C 180,E1 -1173.39,E2 -1173.39} C_VEL
LIN {X 0,Y 594.232,Z 474.384,A -85,B 0,C 180,E1 -1174.749,E2 -1174.749} C_VEL
LIN {X 0,Y 594.279,Z 469.608,A -85,B 0,C 180,E1 -1176.11,E2 -1176.11} C_VEL
LIN {X 0,Y 594.287,Z 463.424,A -85,B 0,C 180,E1 -1177.475,E2 -1177.475} C_VEL
LIN {X 0,Y 594.331,Z 455.651,A -85,B 0,C 180,E1 -1178.843,E2 -1178.843} C_VEL
LIN {X 0,Y 594.387,Z 447.37,A -85,B 0,C 180,E1 -1180.044,E2 -1180.044} C_VEL
LIN {X 0,Y 594.433,Z 437.559,A -85,B 0,C 180,E1 -1181.231,E2 -1181.231} C_VEL
LIN {X 0,Y 594.53,Z 427.191,A -85,B 0,C 180,E1 -1182.285,E2 -1182.285} C_VEL
LIN {X 0,Y 594.581,Z 415.017,A -85,B 0,C 180,E1 -1183.326,E2 -1183.326} C_VEL
LIN {X 0,Y 594.694,Z 403.072,A -85,B 0,C 180,E1 -1184.178,E2 -1184.178} C_VEL
LIN {X 0,Y 594.764,Z 389.521,A -85,B 0,C 180,E1 -1184.98,E2 -1184.98} C_VEL
LIN {X 0,Y 594.883,Z 374.837,A -85,B 0,C 180,E1 -1185.679,E2 -1185.679} C_VEL
LIN {X 0,Y 594.973,Z 360.616,A -85,B 0,C 180,E1 -1186.204,E2 -1186.204} C_VEL
LIN {X 0,Y 595.055,Z 346.035,A -85,B 0,C 180,E1 -1186.605,E2 -1186.605} C_VEL
LIN {X 0,Y 595.099,Z 331.668,A -85,B 0,C 180,E1 -1186.871,E2 -1186.871} C_VEL
LIN {X 0,Y 595.294,Z 173.444,A -85,B 0,C 180,E1 -1188.837,E2 -1188.837} C_VEL
LIN {X 0,Y 594.723,Z 170.178,A -85,B 0,C 180,E1 -1188.92,E2 -1188.92} C_VEL
LIN {X 0,Y 594.844,Z 145.832,A -85,B 0,C 180,E1 -1191.849,E2 -1191.849} C_VEL
LIN {X 0,Y 594.958,Z 124.966,A -85,B 0,C 180,E1 -1194.421,E2 -1194.421} C_VEL
LIN {X 0,Y 594.374,Z 122.128,A -85,B 0,C 180,E1 -1194.842,E2 -1194.842} C_VEL
LIN {X 0,Y 594.387,Z 122.067,A -85,B 0,C 180,E1 -1197.527,E2 -1197.527} C_VEL
LIN {X 0,Y 594.387,Z 122.072,A -85,B 0,C 180,E1 -1200.328,E2 -1200.328} C_VEL
LIN {X 0,Y 594.378,Z 122.066,A -85,B 0,C 180,E1 -1202.95,E2 -1202.95} C_VEL
LIN {X 0,Y 594.348,Z 122.071,A -85,B 0,C 180,E1 -1205.409,E2 -1205.409} C_VEL
LIN {X 0,Y 594.386,Z 122.075,A -85,B 0,C 180,E1 -1207.941,E2 -1207.941} C_VEL
LIN {X 0,Y 594.377,Z 122.066,A -85,B 0,C 180,E1 -1210.822,E2 -1210.822} C_VEL
LIN {X 0,Y 594.367,Z 122.07,A -85,B 0,C 180,E1 -1213.3,E2 -1213.3} C_VEL
LIN {X 0,Y 594.369,Z 122.071,A -85,B 0,C 180,E1 -1216.161,E2 -1216.161} C_VEL
LIN {X 0,Y 594.378,Z 122.065,A -85,B 0,C 180,E1 -1218.536,E2 -1218.536} C_VEL
LIN {X 0,Y 594.382,Z 122.07,A -85,B 0,C 180,E1 -1221.296,E2 -1221.296} C_VEL
LIN {X 0,Y 594.35,Z 122.075,A -85,B 0,C 180,E1 -1223.755,E2 -1223.755} C_VEL
LIN {X 0,Y 594.365,Z 122.065,A -85,B 0,C 180,E1 -1226.238,E2 -1226.238} C_VEL
LIN {X 0,Y 594.369,Z 122.066,A -85,B 0,C 180,E1 -1228.65,E2 -1228.65} C_VEL
LIN {X 0,Y 594.384,Z 122.071,A -85,B 0,C 180,E1 -1231.042,E2 -1231.042} C_VEL
LIN {X 0,Y 594.378,Z 122.066,A -85,B 0,C 180,E1 -1233.979,E2 -1233.979} C_VEL
LIN {X 0,Y 594.369,Z 122.067,A -85,B 0,C 180,E1 -1236.295,E2 -1236.295} C_VEL
LIN {X 0,Y 594.397,Z 122.071,A -85,B 0,C 180,E1 -1239.224,E2 -1239.224} C_VEL
LIN {X 0,Y 594.34,Z 122.071,A -85,B 0,C 180,E1 -1242.095,E2 -1242.095} C_VEL
LIN {X 0,Y 594.361,Z 122.068,A -85,B 0,C 180,E1 -1244.219,E2 -1244.219} C_VEL
LIN {X 0,Y 594.357,Z 122.076,A -85,B 0,C 180,E1 -1247.017,E2 -1247.017} C_VEL
LIN {X 0,Y 594.386,Z 122.064,A -85,B 0,C 180,E1 -1249.784,E2 -1249.784} C_VEL
LIN {X 0,Y 594.394,Z 122.071,A -85,B 0,C 180,E1 -1252.527,E2 -1252.527} C_VEL
LIN {X 0,Y 594.371,Z 122.068,A -85,B 0,C 180,E1 -1255.252,E2 -1255.252} C_VEL
LIN {X 0,Y 594.404,Z 122.064,A -85,B 0,C 180,E1 -1257.967,E2 -1257.967} C_VEL
LIN {X 0,Y 594.416,Z 122.067,A -85,B 0,C 180,E1 -1260.678,E2 -1260.678} C_VEL
LIN {X 0,Y 594.331,Z 122.071,A -85,B 0,C 180,E1 -1263.39,E2 -1263.39} C_VEL
LIN {X 0,Y 594.385,Z 122.072,A -85,B 0,C 180,E1 -1266.109,E2 -1266.109} C_VEL
LIN {X 0,Y 594.367,Z 122.068,A -85,B 0,C 180,E1 -1268.842,E2 -1268.842} C_VEL
LIN {X 0,Y 594.377,Z 122.068,A -85,B 0,C 180,E1 -1271.596,E2 -1271.596} C_VEL
LIN {X 0,Y 594.382,Z 122.07,A -85,B 0,C 180,E1 -1274.377,E2 -1274.377} C_VEL
LIN {X 0,Y 594.337,Z 122.071,A -85,B 0,C 180,E1 -1275.312,E2 -1275.312} C_VEL
LIN {X 0,Y 593.67,Z 122.162,A -85,B 0,C 180,E1 -1275.878,E2 -1275.878} C_VEL
LIN {X 0,Y 590.806,Z 122.522,A -85,B 0,C 180,E1 -1276.795,E2 -1276.795} C_VEL
LIN {X 0,Y 588.393,Z 122.823,A -85,B 0,C 180,E1 -1277.533,E2 -1277.533} C_VEL
LIN {X 0,Y 587.367,Z 122.947,A -85,B 0,C 180,E1 -1278.103,E2 -1278.103} C_VEL
LIN {X 0,Y 587.289,Z 122.953,A -85,B 0,C 180,E1 -1278.296,E2 -1278.296} C_VEL
LIN {X 0,Y 587.333,Z 122.943,A -85,B 0,C 180,E1 -1281.038,E2 -1281.038} C_VEL
LIN {X 0,Y 587.297,Z 122.954,A -85,B 0,C 180,E1 -1284.008,E2 -1284.008} C_VEL
LIN {X 0,Y 587.306,Z 122.949,A -85,B 0,C 180,E1 -1286.28,E2 -1286.28} C_VEL
LIN {X 0,Y 587.341,Z 122.945,A -85,B 0,C 180,E1 -1289.132,E2 -1289.132} C_VEL
LIN {X 0,Y 587.315,Z 122.948,A -85,B 0,C 180,E1 -1291.831,E2 -1291.831} C_VEL
LIN {X 0,Y 587.329,Z 122.944,A -85,B 0,C 180,E1 -1294.345,E2 -1294.345} C_VEL
LIN {X 0,Y 587.338,Z 122.949,A -85,B 0,C 180,E1 -1297.608,E2 -1297.608} C_VEL
LIN {X 0,Y 587.294,Z 122.945,A -85,B 0,C 180,E1 -1300.256,E2 -1300.256} C_VEL
LIN {X 0,Y 587.29,Z 122.956,A -85,B 0,C 180,E1 -1303.115,E2 -1303.115} C_VEL
LIN {X 0,Y 587.298,Z 122.947,A -85,B 0,C 180,E1 -1306.047,E2 -1306.047} C_VEL
LIN {X 0,Y 587.331,Z 122.951,A -85,B 0,C 180,E1 -1308.926,E2 -1308.926} C_VEL
LIN {X 0,Y 587.311,Z 122.95,A -85,B 0,C 180,E1 -1311.519,E2 -1311.519} C_VEL
LIN {X 0,Y 587.265,Z 122.952,A -85,B 0,C 180,E1 -1314.098,E2 -1314.098} C_VEL
LIN {X 0,Y 587.331,Z 122.953,A -85,B 0,C 180,E1 -1316.89,E2 -1316.89} C_VEL
LIN {X 0,Y 587.292,Z 122.945,A -85,B 0,C 180,E1 -1319.827,E2 -1319.827} C_VEL
LIN {X 0,Y 587.309,Z 122.951,A -85,B 0,C 180,E1 -1322.953,E2 -1322.953} C_VEL
LIN {X 0,Y 587.331,Z 123,A -85,B 0,C 180,E1 -1325.912,E2 -1325.912} C_VEL
LIN {X 0,Y 587.412,Z 123.53,A -85,B 0,C 180,E1 -1326.091,E2 -1326.091} C_VEL
LIN {X 0,Y 588.004,Z 127.007,A -85,B 0,C 180,E1 -1326.583,E2 -1326.583} C_VEL
LIN {X 0,Y 587.853,Z 148.302,A -85,B 0,C 180,E1 -1329.348,E2 -1329.348} C_VEL
LIN {X 0,Y 587.744,Z 160.733,A -85,B 0,C 180,E1 -1330.906,E2 -1330.906} C_VEL
LIN {X 0,Y 588.616,Z 165.722,A -85,B 0,C 180,E1 -1331.015,E2 -1331.015} C_VEL
LIN {X 0,Y 588.296,Z 326.469,A -85,B 0,C 180,E1 -1333.046,E2 -1333.046} C_VEL
LIN {X 0,Y 588.208,Z 342.478,A -85,B 0,C 180,E1 -1333.403,E2 -1333.403} C_VEL
LIN {X 0,Y 588.105,Z 357.036,A -85,B 0,C 180,E1 -1333.868,E2 -1333.868} C_VEL
LIN {X 0,Y 587.958,Z 371.704,A -85,B 0,C 180,E1 -1334.487,E2 -1334.487} C_VEL
LIN {X 0,Y 587.844,Z 385.01,A -85,B 0,C 180,E1 -1335.194,E2 -1335.194} C_VEL
LIN {X 0,Y 587.735,Z 398.176,A -85,B 0,C 180,E1 -1336.047,E2 -1336.047} C_VEL
LIN {X 0,Y 587.558,Z 410.866,A -85,B 0,C 180,E1 -1337.04,E2 -1337.04} C_VEL
LIN {X 0,Y 587.472,Z 422.068,A -85,B 0,C 180,E1 -1338.091,E2 -1338.091} C_VEL
LIN {X 0,Y 587.383,Z 432.951,A -85,B 0,C 180,E1 -1339.312,E2 -1339.312} C_VEL
LIN {X 0,Y 587.285,Z 441.994,A -85,B 0,C 180,E1 -1340.529,E2 -1340.529} C_VEL
LIN {X 0,Y 587.258,Z 449.487,A -85,B 0,C 180,E1 -1341.743,E2 -1341.743} C_VEL
LIN {X 0,Y 587.208,Z 456.492,A -85,B 0,C 180,E1 -1343.126,E2 -1343.126} C_VEL
LIN {X 0,Y 587.198,Z 462.001,A -85,B 0,C 180,E1 -1344.506,E2 -1344.506} C_VEL
LIN {X 0,Y 587.169,Z 466.173,A -85,B 0,C 180,E1 -1345.882,E2 -1345.882} C_VEL
LIN {X 0,Y 587.127,Z 469.113,A -85,B 0,C 180,E1 -1347.256,E2 -1347.256} C_VEL
LIN {X 0,Y 587.143,Z 470.88,A -85,B 0,C 180,E1 -1348.628,E2 -1348.628} C_VEL
LIN {X 0,Y 587.135,Z 471.496,A -85,B 0,C 180,E1 -1350,E2 -1350} C_VEL
LIN {X 0,Y 587.145,Z 470.943,A -85,B 0,C 180,E1 -1351.372,E2 -1351.372} C_VEL
LIN {X 0,Y 587.129,Z 469.26,A -85,B 0,C 180,E1 -1352.744,E2 -1352.744} C_VEL
LIN {X 0,Y 587.169,Z 466.406,A -85,B 0,C 180,E1 -1354.118,E2 -1354.118} C_VEL
LIN {X 0,Y 587.198,Z 462.323,A -85,B 0,C 180,E1 -1355.495,E2 -1355.495} C_VEL
LIN {X 0,Y 587.208,Z 456.912,A -85,B 0,C 180,E1 -1356.874,E2 -1356.874} C_VEL
LIN {X 0,Y 587.254,Z 450.012,A -85,B 0,C 180,E1 -1358.257,E2 -1358.257} C_VEL
LIN {X 0,Y 587.286,Z 441.408,A -85,B 0,C 180,E1 -1359.645,E2 -1359.645} C_VEL
LIN {X 0,Y 587.367,Z 432.258,A -85,B 0,C 180,E1 -1360.863,E2 -1360.863} C_VEL
LIN {X 0,Y 587.447,Z 422.93,A -85,B 0,C 180,E1 -1361.91,E2 -1361.91} C_VEL
LIN {X 0,Y 587.589,Z 410.888,A -85,B 0,C 180,E1 -1363.048,E2 -1363.048} C_VEL
LIN {X 0,Y 587.711,Z 397.794,A -85,B 0,C 180,E1 -1364.069,E2 -1364.069} C_VEL
LIN {X 0,Y 587.807,Z 385.035,A -85,B 0,C 180,E1 -1364.896,E2 -1364.896} C_VEL
LIN {X 0,Y 587.979,Z 371.73,A -85,B 0,C 180,E1 -1365.601,E2 -1365.601} C_VEL
LIN {X 0,Y 588.085,Z 357.052,A -85,B 0,C 180,E1 -1366.221,E2 -1366.221} C_VEL
LIN {X 0,Y 588.223,Z 341.284,A -85,B 0,C 180,E1 -1366.72,E2 -1366.72} C_VEL
LIN {X 0,Y 588.294,Z 326.368,A -85,B 0,C 180,E1 -1367.046,E2 -1367.046} C_VEL
LIN {X 0,Y 588.603,Z 165.294,A -85,B 0,C 180,E1 -1369.081,E2 -1369.081} C_VEL
LIN {X 0,Y 587.752,Z 160.712,A -85,B 0,C 180,E1 -1369.184,E2 -1369.184} C_VEL
LIN {X 0,Y 587.892,Z 141.968,A -85,B 0,C 180,E1 -1371.559,E2 -1371.559} C_VEL
LIN {X 0,Y 587.977,Z 126.271,A -85,B 0,C 180,E1 -1373.605,E2 -1373.605} C_VEL
LIN {X 0,Y 587.327,Z 123.102,A -85,B 0,C 180,E1 -1374.088,E2 -1374.088} C_VEL
LIN {X 0,Y 587.295,Z 122.952,A -85,B 0,C 180,E1 -1377.048,E2 -1377.048} C_VEL
LIN {X 0,Y 587.29,Z 122.946,A -85,B 0,C 180,E1 -1380.173,E2 -1380.173} C_VEL
LIN {X 0,Y 587.304,Z 122.95,A -85,B 0,C 180,E1 -1382.581,E2 -1382.581} C_VEL
LIN {X 0,Y 587.292,Z 122.958,A -85,B 0,C 180,E1 -1385.058,E2 -1385.058} C_VEL
LIN {X 0,Y 587.312,Z 122.947,A -85,B 0,C 180,E1 -1387.835,E2 -1387.835} C_VEL
LIN {X 0,Y 587.291,Z 122.948,A -85,B 0,C 180,E1 -1390.256,E2 -1390.256} C_VEL
LIN {X 0,Y 587.288,Z 122.954,A -85,B 0,C 180,E1 -1393.115,E2 -1393.115} C_VEL
LIN {X 0,Y 587.299,Z 122.948,A -85,B 0,C 180,E1 -1396.047,E2 -1396.047} C_VEL
LIN {X 0,Y 587.31,Z 122.95,A -85,B 0,C 180,E1 -1398.928,E2 -1398.928} C_VEL
LIN {X 0,Y 587.303,Z 122.947,A -85,B 0,C 180,E1 -1401.518,E2 -1401.518} C_VEL
LIN {X 0,Y 587.275,Z 122.954,A -85,B 0,C 180,E1 -1404.099,E2 -1404.099} C_VEL
LIN {X 0,Y 587.333,Z 122.944,A -85,B 0,C 180,E1 -1406.89,E2 -1406.89} C_VEL
LIN {X 0,Y 587.317,Z 122.943,A -85,B 0,C 180,E1 -1409.494,E2 -1409.494} C_VEL
LIN {X 0,Y 587.29,Z 122.956,A -85,B 0,C 180,E1 -1412.179,E2 -1412.179} C_VEL
LIN {X 0,Y 587.325,Z 122.95,A -85,B 0,C 180,E1 -1414.483,E2 -1414.483} C_VEL
LIN {X 0,Y 587.308,Z 122.948,A -85,B 0,C 180,E1 -1417.485,E2 -1417.485} C_VEL
LIN {X 0,Y 587.309,Z 122.949,A -85,B 0,C 180,E1 -1419.694,E2 -1419.694} C_VEL
LIN {X 0,Y 587.286,Z 122.956,A -85,B 0,C 180,E1 -1421.872,E2 -1421.872} C_VEL
LIN {X 0,Y 587.307,Z 122.946,A -85,B 0,C 180,E1 -1424.736,E2 -1424.736} C_VEL
LIN {X 0,Y 587.285,Z 122.949,A -85,B 0,C 180,E1 -1426.858,E2 -1426.858} C_VEL
LIN {X 0,Y 587.334,Z 122.951,A -85,B 0,C 180,E1 -1429.66,E2 -1429.66} C_VEL
LIN {X 0,Y 587.345,Z 122.943,A -85,B 0,C 180,E1 -1432.437,E2 -1432.437} C_VEL
LIN {X 0,Y 587.346,Z 122.945,A -85,B 0,C 180,E1 -1435.195,E2 -1435.195} C_VEL
LIN {X 0,Y 587.375,Z 122.942,A -85,B 0,C 180,E1 -1437.943,E2 -1437.943} C_VEL
LIN {X 0,Y 587.37,Z 122.939,A -85,B 0,C 180,E1 -1440.685,E2 -1440.685} C_VEL
LIN {X 0,Y 587.325,Z 122.953,A -85,B 0,C 180,E1 -1443.43,E2 -1443.43} C_VEL
LIN {X 0,Y 587.331,Z 122.944,A -85,B 0,C 180,E1 -1446.182,E2 -1446.182} C_VEL
LIN {X 0,Y 587.339,Z 122.942,A -85,B 0,C 180,E1 -1448.256,E2 -1448.256} C_VEL
LIN {X 0,Y 587.352,Z 122.949,A -85,B 0,C 180,E1 -1451.134,E2 -1451.134} C_VEL
LIN {X 0,Y 587.335,Z 122.943,A -85,B 0,C 180,E1 -1454.247,E2 -1454.247} C_VEL
LIN {X 0,Y 587.334,Z 122.948,A -85,B 0,C 180,E1 -1456.808,E2 -1456.808} C_VEL
LIN {X 0,Y 587.31,Z 122.948,A -85,B 0,C 180,E1 -1459.576,E2 -1459.576} C_VEL
LIN {X 0,Y 587.315,Z 122.945,A -85,B 0,C 180,E1 -1461.775,E2 -1461.775} C_VEL
LIN {X 0,Y 587.314,Z 122.955,A -85,B 0,C 180,E1 -1464.76,E2 -1464.76} C_VEL
LIN {X 0,Y 587.33,Z 122.949,A -85,B 0,C 180,E1 -1467.046,E2 -1467.046} C_VEL
LIN {X 0,Y 587.341,Z 122.943,A -85,B 0,C 180,E1 -1469.38,E2 -1469.38} C_VEL
LIN {X 0,Y 587.342,Z 122.94,A -85,B 0,C 180,E1 -1471.835,E2 -1471.835} C_VEL
LIN {X 0,Y 587.344,Z 122.945,A -85,B 0,C 180,E1 -1474.347,E2 -1474.347} C_VEL
LIN {X 0,Y 587.344,Z 122.943,A -85,B 0,C 180,E1 -1477.608,E2 -1477.608} C_VEL
LIN {X 0,Y 587.312,Z 122.953,A -85,B 0,C 180,E1 -1480.254,E2 -1480.254} C_VEL
LIN {X 0,Y 587.318,Z 122.946,A -85,B 0,C 180,E1 -1483.118,E2 -1483.118} C_VEL
LIN {X 0,Y 587.314,Z 122.952,A -85,B 0,C 180,E1 -1486.048,E2 -1486.048} C_VEL
LIN {X 0,Y 587.337,Z 122.944,A -85,B 0,C 180,E1 -1488.925,E2 -1488.925} C_VEL
LIN {X 0,Y 587.332,Z 122.946,A -85,B 0,C 180,E1 -1491.521,E2 -1491.521} C_VEL
LIN {X 0,Y 587.291,Z 122.957,A -85,B 0,C 180,E1 -1494.1,E2 -1494.1} C_VEL
LIN {X 0,Y 587.336,Z 122.943,A -85,B 0,C 180,E1 -1496.603,E2 -1496.603} C_VEL
LIN {X 0,Y 587.337,Z 122.946,A -85,B 0,C 180,E1 -1499.49,E2 -1499.49} C_VEL
LIN {X 0,Y 587.352,Z 122.944,A -85,B 0,C 180,E1 -1502.307,E2 -1502.307} C_VEL
LIN {X 0,Y 587.36,Z 123.073,A -85,B 0,C 180,E1 -1504.982,E2 -1504.982} C_VEL
LIN {X 0,Y 588.08,Z 126.418,A -85,B 0,C 180,E1 -1505.458,E2 -1505.458} C_VEL
LIN {X 0,Y 587.971,Z 144.341,A -85,B 0,C 180,E1 -1507.697,E2 -1507.697} C_VEL
LIN {X 0,Y 587.757,Z 167.787,A -85,B 0,C 180,E1 -1510.572,E2 -1510.572} C_VEL
LIN {X 0,Y 587.81,Z 170.569,A -85,B 0,C 180,E1 -1510.87,E2 -1510.87} C_VEL
LIN {X 0,Y 588.598,Z 175.229,A -85,B 0,C 180,E1 -1510.963,E2 -1510.963} C_VEL
LIN {X 0,Y 588.315,Z 336.067,A -85,B 0,C 180,E1 -1512.994,E2 -1512.994} C_VEL
LIN {X 0,Y 588.223,Z 351.704,A -85,B 0,C 180,E1 -1513.337,E2 -1513.337} C_VEL
LIN {X 0,Y 588.083,Z 367.041,A -85,B 0,C 180,E1 -1513.823,E2 -1513.823} C_VEL
LIN {X 0,Y 587.979,Z 380.766,A -85,B 0,C 180,E1 -1514.399,E2 -1514.399} C_VEL
LIN {X 0,Y 587.834,Z 394.24,A -85,B 0,C 180,E1 -1515.105,E2 -1515.105} C_VEL
LIN {X 0,Y 587.741,Z 407.114,A -85,B 0,C 180,E1 -1515.929,E2 -1515.929} C_VEL
LIN {X 0,Y 587.582,Z 419.287,A -85,B 0,C 180,E1 -1516.864,E2 -1516.864} C_VEL
LIN {X 0,Y 587.454,Z 430.748,A -85,B 0,C 180,E1 -1517.915,E2 -1517.915} C_VEL
LIN {X 0,Y 587.348,Z 440.39,A -85,B 0,C 180,E1 -1518.963,E2 -1518.963} C_VEL
LIN {X 0,Y 587.305,Z 449.856,A -85,B 0,C 180,E1 -1520.182,E2 -1520.182} C_VEL
LIN {X 0,Y 587.265,Z 457.732,A -85,B 0,C 180,E1 -1521.397,E2 -1521.397} C_VEL
LIN {X 0,Y 587.215,Z 465.088,A -85,B 0,C 180,E1 -1522.781,E2 -1522.781} C_VEL
LIN {X 0,Y 587.227,Z 470.923,A -85,B 0,C 180,E1 -1524.161,E2 -1524.161} C_VEL
LIN {X 0,Y 587.136,Z 474.384,A -85,B 0,C 180,E1 -1525.194,E2 -1525.194} C_VEL
LIN {X 0,Y 587.18,Z 477.888,A -85,B 0,C 180,E1 -1526.569,E2 -1526.569} C_VEL
LIN {X 0,Y 587.14,Z 480.193,A -85,B 0,C 180,E1 -1527.942,E2 -1527.942} C_VEL
LIN {X 0,Y 587.135,Z 481.35,A -85,B 0,C 180,E1 -1529.314,E2 -1529.314} C_VEL
LIN {X 0,Y 587.135,Z 481.349,A -85,B 0,C 180,E1 -1530.686,E2 -1530.686} C_VEL
LIN {X 0,Y 587.14,Z 480.192,A -85,B 0,C 180,E1 -1532.058,E2 -1532.058} C_VEL
LIN {X 0,Y 587.18,Z 477.886,A -85,B 0,C 180,E1 -1533.431,E2 -1533.431} C_VEL
LIN {X 0,Y 587.136,Z 474.385,A -85,B 0,C 180,E1 -1534.806,E2 -1534.806} C_VEL
LIN {X 0,Y 587.18,Z 469.608,A -85,B 0,C 180,E1 -1536.184,E2 -1536.184} C_VEL
LIN {X 0,Y 587.23,Z 463.424,A -85,B 0,C 180,E1 -1537.565,E2 -1537.565} C_VEL
LIN {X 0,Y 587.266,Z 455.65,A -85,B 0,C 180,E1 -1538.95,E2 -1538.95} C_VEL
LIN {X 0,Y 587.351,Z 447.369,A -85,B 0,C 180,E1 -1540.166,E2 -1540.166} C_VEL
LIN {X 0,Y 587.4,Z 437.395,A -85,B 0,C 180,E1 -1541.386,E2 -1541.386} C_VEL
LIN {X 0,Y 587.522,Z 427.19,A -85,B 0,C 180,E1 -1542.434,E2 -1542.434} C_VEL
LIN {X 0,Y 587.629,Z 415.018,A -85,B 0,C 180,E1 -1543.487,E2 -1543.487} C_VEL
LIN {X 0,Y 587.774,Z 402.058,A -85,B 0,C 180,E1 -1544.416,E2 -1544.416} C_VEL
LIN {X 0,Y 587.89,Z 387.867,A -85,B 0,C 180,E1 -1545.248,E2 -1545.248} C_VEL
LIN {X 0,Y 588.033,Z 373.796,A -85,B 0,C 180,E1 -1545.911,E2 -1545.911} C_VEL
LIN {X 0,Y 588.169,Z 359.303,A -85,B 0,C 180,E1 -1546.442,E2 -1546.442} C_VEL
LIN {X 0,Y 588.273,Z 344.193,A -85,B 0,C 180,E1 -1546.847,E2 -1546.847} C_VEL
LIN {X 0,Y 588.321,Z 329.156,A -85,B 0,C 180,E1 -1547.109,E2 -1547.109} C_VEL
LIN {X 0,Y 588.482,Z 173.994,A -85,B 0,C 180,E1 -1549.057,E2 -1549.057} C_VEL
LIN {X 0,Y 587.785,Z 170.2,A -85,B 0,C 180,E1 -1549.151,E2 -1549.151} C_VEL
LIN {X 0,Y 587.968,Z 147.322,A -85,B 0,C 180,E1 -1551.934,E2 -1551.934} C_VEL
LIN {X 0,Y 588.132,Z 128.093,A -85,B 0,C 180,E1 -1554.329,E2 -1554.329} C_VEL
LIN {X 0,Y 587.777,Z 124.96,A -85,B 0,C 180,E1 -1554.739,E2 -1554.739} C_VEL
LIN {X 0,Y 587.345,Z 123.011,A -85,B 0,C 180,E1 -1555.042,E2 -1555.042} C_VEL
LIN {X 0,Y 587.347,Z 122.945,A -85,B 0,C 180,E1 -1557.818,E2 -1557.818} C_VEL
LIN {X 0,Y 587.337,Z 122.946,A -85,B 0,C 180,E1 -1560.51,E2 -1560.51} C_VEL
LIN {X 0,Y 587.335,Z 122.944,A -85,B 0,C 180,E1 -1563.397,E2 -1563.397} C_VEL
LIN {X 0,Y 587.291,Z 122.957,A -85,B 0,C 180,E1 -1565.9,E2 -1565.9} C_VEL
LIN {X 0,Y 587.333,Z 122.945,A -85,B 0,C 180,E1 -1568.479,E2 -1568.479} C_VEL
LIN {X 0,Y 587.337,Z 122.944,A -85,B 0,C 180,E1 -1571.157,E2 -1571.157} C_VEL
LIN {X 0,Y 587.313,Z 122.95,A -85,B 0,C 180,E1 -1574.112,E2 -1574.112} C_VEL
LIN {X 0,Y 587.317,Z 122.947,A -85,B 0,C 180,E1 -1576.994,E2 -1576.994} C_VEL
LIN {X 0,Y 587.312,Z 122.953,A -85,B 0,C 180,E1 -1579.746,E2 -1579.746} C_VEL
LIN {X 0,Y 587.344,Z 122.943,A -85,B 0,C 180,E1 -1582.392,E2 -1582.392} C_VEL
LIN {X 0,Y 587.343,Z 122.946,A -85,B 0,C 180,E1 -1585.653,E2 -1585.653} C_VEL
LIN {X 0,Y 587.34,Z 122.941,A -85,B 0,C 180,E1 -1588.231,E2 -1588.231} C_VEL
LIN {X 0,Y 587.349,Z 122.945,A -85,B 0,C 180,E1 -1590.867,E2 -1590.867} C_VEL
LIN {X 0,Y 587.339,Z 122.944,A -85,B 0,C 180,E1 -1593.824,E2 -1593.824} C_VEL
LIN {X 0,Y 587.316,Z 122.946,A -85,B 0,C 180,E1 -1595.993,E2 -1595.993} C_VEL
LIN {X 0,Y 587.316,Z 122.945,A -85,B 0,C 180,E1 -1598.226,E2 -1598.226} C_VEL
LIN {X 0,Y 587.344,Z 122.951,A -85,B 0,C 180,E1 -1601.151,E2 -1601.151} C_VEL
LIN {X 0,Y 587.314,Z 122.945,A -85,B 0,C 180,E1 -1604.025,E2 -1604.025} C_VEL
LIN {X 0,Y 587.31,Z 122.956,A -85,B 0,C 180,E1 -1606.858,E2 -1606.858} C_VEL
LIN {X 0,Y 587.334,Z 122.942,A -85,B 0,C 180,E1 -1609.66,E2 -1609.66} C_VEL
LIN {X 0,Y 587.363,Z 122.945,A -85,B 0,C 180,E1 -1612.437,E2 -1612.437} C_VEL
LIN {X 0,Y 587.345,Z 122.943,A -85,B 0,C 180,E1 -1615.195,E2 -1615.195} C_VEL
LIN {X 0,Y 587.373,Z 122.939,A -85,B 0,C 180,E1 -1617.943,E2 -1617.943} C_VEL
LIN {X 0,Y 587.387,Z 122.942,A -85,B 0,C 180,E1 -1620.686,E2 -1620.686} C_VEL
LIN {X 0,Y 587.362,Z 122.944,A -85,B 0,C 180,E1 -1622.743,E2 -1622.743} C_VEL
LIN {X 0,Y 587.345,Z 122.942,A -85,B 0,C 180,E1 -1625.493,E2 -1625.493} C_VEL
LIN {X 0,Y 587.362,Z 122.948,A -85,B 0,C 180,E1 -1628.255,E2 -1628.255} C_VEL
LIN {X 0,Y 587.333,Z 122.944,A -85,B 0,C 180,E1 -1631.124,E2 -1631.124} C_VEL
LIN {X 0,Y 587.354,Z 122.946,A -85,B 0,C 180,E1 -1633.846,E2 -1633.846} C_VEL
LIN {X 0,Y 587.289,Z 122.95,A -85,B 0,C 180,E1 -1636.794,E2 -1636.794} C_VEL
LIN {X 0,Y 587.289,Z 122.953,A -85,B 0,C 180,E1 -1638.296,E2 -1638.296} C_VEL
LIN {X 0,Y 586.649,Z 123.03,A -85,B 0,C 180,E1 -1638.868,E2 -1638.868} C_VEL
LIN {X 0,Y 583.841,Z 123.386,A -85,B 0,C 180,E1 -1639.797,E2 -1639.797} C_VEL
LIN {X 0,Y 581.439,Z 123.682,A -85,B 0,C 180,E1 -1640.544,E2 -1640.544} C_VEL
LIN {X 0,Y 580.383,Z 123.81,A -85,B 0,C 180,E1 -1641.12,E2 -1641.12} C_VEL
LIN {X 0,Y 580.284,Z 123.823,A -85,B 0,C 180,E1 -1641.316,E2 -1641.316} C_VEL
LIN {X 0,Y 580.256,Z 123.831,A -85,B 0,C 180,E1 -1643.559,E2 -1643.559} C_VEL
LIN {X 0,Y 580.265,Z 123.826,A -85,B 0,C 180,E1 -1646.328,E2 -1646.328} C_VEL
LIN {X 0,Y 580.276,Z 123.827,A -85,B 0,C 180,E1 -1649.305,E2 -1649.305} C_VEL
LIN {X 0,Y 580.284,Z 123.818,A -85,B 0,C 180,E1 -1652.202,E2 -1652.202} C_VEL
LIN {X 0,Y 580.276,Z 123.822,A -85,B 0,C 180,E1 -1654.697,E2 -1654.697} C_VEL
LIN {X 0,Y 580.286,Z 123.829,A -85,B 0,C 180,E1 -1657.27,E2 -1657.27} C_VEL
LIN {X 0,Y 580.275,Z 123.819,A -85,B 0,C 180,E1 -1660.268,E2 -1660.268} C_VEL
LIN {X 0,Y 580.251,Z 123.827,A -85,B 0,C 180,E1 -1662.709,E2 -1662.709} C_VEL
LIN {X 0,Y 580.251,Z 123.828,A -85,B 0,C 180,E1 -1665.611,E2 -1665.611} C_VEL
LIN {X 0,Y 580.269,Z 123.827,A -85,B 0,C 180,E1 -1668.67,E2 -1668.67} C_VEL
LIN {X 0,Y 580.264,Z 123.831,A -85,B 0,C 180,E1 -1670.964,E2 -1670.964} C_VEL
LIN {X 0,Y 580.238,Z 123.829,A -85,B 0,C 180,E1 -1673.594,E2 -1673.594} C_VEL
LIN {X 0,Y 580.27,Z 123.824,A -85,B 0,C 180,E1 -1676.142,E2 -1676.142} C_VEL
LIN {X 0,Y 580.248,Z 123.833,A -85,B 0,C 180,E1 -1678.613,E2 -1678.613} C_VEL
LIN {X 0,Y 580.245,Z 123.834,A -85,B 0,C 180,E1 -1681.021,E2 -1681.021} C_VEL
LIN {X 0,Y 580.25,Z 123.828,A -85,B 0,C 180,E1 -1683.675,E2 -1683.675} C_VEL
LIN {X 0,Y 580.296,Z 124.043,A -85,B 0,C 180,E1 -1685.826,E2 -1685.826} C_VEL
LIN {X 0,Y 581.14,Z 128.454,A -85,B 0,C 180,E1 -1686.479,E2 -1686.479} C_VEL
LIN {X 0,Y 580.926,Z 148.306,A -85,B 0,C 180,E1 -1689.091,E2 -1689.091} C_VEL
LIN {X 0,Y 580.833,Z 160.716,A -85,B 0,C 180,E1 -1690.668,E2 -1690.668} C_VEL
LIN {X 0,Y 581.896,Z 166.148,A -85,B 0,C 180,E1 -1690.792,E2 -1690.792} C_VEL
LIN {X 0,Y 581.53,Z 326.034,A -85,B 0,C 180,E1 -1692.834,E2 -1692.834} C_VEL
LIN {X 0,Y 581.402,Z 341.724,A -85,B 0,C 180,E1 -1693.181,E2 -1693.181} C_VEL
LIN {X 0,Y 581.249,Z 357.049,A -85,B 0,C 180,E1 -1693.673,E2 -1693.673} C_VEL
LIN {X 0,Y 581.102,Z 371.713,A -85,B 0,C 180,E1 -1694.299,E2 -1694.299} C_VEL
LIN {X 0,Y 580.924,Z 385.023,A -85,B 0,C 180,E1 -1695.013,E2 -1695.013} C_VEL
LIN {X 0,Y 580.792,Z 398.373,A -85,B 0,C 180,E1 -1695.89,E2 -1695.89} C_VEL
LIN {X 0,Y 580.593,Z 410.874,A -85,B 0,C 180,E1 -1696.881,E2 -1696.881} C_VEL
LIN {X 0,Y 580.46,Z 422.073,A -85,B 0,C 180,E1 -1697.945,E2 -1697.945} C_VEL
LIN {X 0,Y 580.337,Z 433.113,A -85,B 0,C 180,E1 -1699.201,E2 -1699.201} C_VEL
LIN {X 0,Y 580.238,Z 441.997,A -85,B 0,C 180,E1 -1700.413,E2 -1700.413} C_VEL
LIN {X 0,Y 580.195,Z 449.49,A -85,B 0,C 180,E1 -1701.642,E2 -1701.642} C_VEL
LIN {X 0,Y 580.139,Z 456.494,A -85,B 0,C 180,E1 -1703.042,E2 -1703.042} C_VEL
LIN {X 0,Y 580.127,Z 462.004,A -85,B 0,C 180,E1 -1704.438,E2 -1704.438} C_VEL
LIN {X 0,Y 580.087,Z 466.174,A -85,B 0,C 180,E1 -1705.831,E2 -1705.831} C_VEL
LIN {X 0,Y 580.038,Z 469.113,A -85,B 0,C 180,E1 -1707.222,E2 -1707.222} C_VEL
LIN {X 0,Y 580.043,Z 470.879,A -85,B 0,C 180,E1 -1708.611,E2 -1708.611} C_VEL
LIN {X 0,Y 580.035,Z 471.496,A -85,B 0,C 180,E1 -1710,E2 -1710} C_VEL
LIN {X 0,Y 580.044,Z 470.942,A -85,B 0,C 180,E1 -1711.389,E2 -1711.389} C_VEL
LIN {X 0,Y 580.04,Z 469.26,A -85,B 0,C 180,E1 -1712.778,E2 -1712.778} C_VEL
LIN {X 0,Y 580.087,Z 466.405,A -85,B 0,C 180,E1 -1714.169,E2 -1714.169} C_VEL
LIN {X 0,Y 580.123,Z 462.321,A -85,B 0,C 180,E1 -1715.562,E2 -1715.562} C_VEL
LIN {X 0,Y 580.139,Z 456.909,A -85,B 0,C 180,E1 -1716.958,E2 -1716.958} C_VEL
LIN {X 0,Y 580.19,Z 450.009,A -85,B 0,C 180,E1 -1718.358,E2 -1718.358} C_VEL
LIN {X 0,Y 580.235,Z 441.403,A -85,B 0,C 180,E1 -1719.763,E2 -1719.763} C_VEL
LIN {X 0,Y 580.308,Z 431.833,A -85,B 0,C 180,E1 -1721.046,E2 -1721.046} C_VEL
LIN {X 0,Y 580.463,Z 421.199,A -85,B 0,C 180,E1 -1722.233,E2 -1722.233} C_VEL
LIN {X 0,Y 580.607,Z 409.824,A -85,B 0,C 180,E1 -1723.296,E2 -1723.296} C_VEL
LIN {X 0,Y 580.76,Z 397.071,A -85,B 0,C 180,E1 -1724.291,E2 -1724.291} C_VEL
LIN {X 0,Y 580.925,Z 383.462,A -85,B 0,C 180,E1 -1725.166,E2 -1725.166} C_VEL
LIN {X 0,Y 581.136,Z 369.785,A -85,B 0,C 180,E1 -1725.88,E2 -1725.88} C_VEL
LIN {X 0,Y 581.272,Z 355.79,A -85,B 0,C 180,E1 -1726.462,E2 -1726.462} C_VEL
LIN {X 0,Y 581.457,Z 340.745,A -85,B 0,C 180,E1 -1726.933,E2 -1726.933} C_VEL
LIN {X 0,Y 581.53,Z 326.319,A -85,B 0,C 180,E1 -1727.251,E2 -1727.251} C_VEL
LIN {X 0,Y 581.79,Z 165.561,A -85,B 0,C 180,E1 -1729.309,E2 -1729.309} C_VEL
LIN {X 0,Y 580.839,Z 160.525,A -85,B 0,C 180,E1 -1729.433,E2 -1729.433} C_VEL
LIN {X 0,Y 581.091,Z 137.631,A -85,B 0,C 180,E1 -1732.394,E2 -1732.394} C_VEL
LIN {X 0,Y 581.065,Z 127.715,A -85,B 0,C 180,E1 -1733.713,E2 -1733.713} C_VEL
LIN {X 0,Y 580.274,Z 123.95,A -85,B 0,C 180,E1 -1734.294,E2 -1734.294} C_VEL
LIN {X 0,Y 580.231,Z 123.831,A -85,B 0,C 180,E1 -1736.626,E2 -1736.626} C_VEL
LIN {X 0,Y 580.245,Z 123.833,A -85,B 0,C 180,E1 -1739.299,E2 -1739.299} C_VEL
LIN {X 0,Y 580.276,Z 123.824,A -85,B 0,C 180,E1 -1742.202,E2 -1742.202} C_VEL
LIN {X 0,Y 580.269,Z 123.827,A -85,B 0,C 180,E1 -1744.698,E2 -1744.698} C_VEL
LIN {X 0,Y 580.281,Z 123.829,A -85,B 0,C 180,E1 -1747.27,E2 -1747.27} C_VEL
LIN {X 0,Y 580.272,Z 123.822,A -85,B 0,C 180,E1 -1750.268,E2 -1750.268} C_VEL
LIN {X 0,Y 580.25,Z 123.833,A -85,B 0,C 180,E1 -1752.709,E2 -1752.709} C_VEL
LIN {X 0,Y 580.252,Z 123.826,A -85,B 0,C 180,E1 -1755.611,E2 -1755.611} C_VEL
LIN {X 0,Y 580.24,Z 123.829,A -85,B 0,C 180,E1 -1758.228,E2 -1758.228} C_VEL
LIN {X 0,Y 580.261,Z 123.829,A -85,B 0,C 180,E1 -1760.964,E2 -1760.964} C_VEL
LIN {X 0,Y 580.243,Z 123.827,A -85,B 0,C 180,E1 -1763.594,E2 -1763.594} C_VEL
LIN {X 0,Y 580.274,Z 123.826,A -85,B 0,C 180,E1 -1766.142,E2 -1766.142} C_VEL
LIN {X 0,Y 580.267,Z 123.828,A -85,B 0,C 180,E1 -1768.614,E2 -1768.614} C_VEL
LIN {X 0,Y 580.278,Z 123.824,A -85,B 0,C 180,E1 -1771.023,E2 -1771.023} C_VEL
LIN {X 0,Y 580.263,Z 123.832,A -85,B 0,C 180,E1 -1774.15,E2 -1774.15} C_VEL
LIN {X 0,Y 580.28,Z 123.822,A -85,B 0,C 180,E1 -1777.197,E2 -1777.197} C_VEL
LIN {X 0,Y 580.276,Z 123.831,A -85,B 0,C 180,E1 -1780.177,E2 -1780.177} C_VEL
LIN {X 0,Y 580.237,Z 123.828,A -85,B 0,C 180,E1 -1783.112,E2 -1783.112} C_VEL
LIN {X 0,Y 580.314,Z 123.826,A -85,B 0,C 180,E1 -1785.983,E2 -1785.983} C_VEL
LIN {X 0,Y 580.309,Z 123.819,A -85,B 0,C 180,E1 -1788.827,E2 -1788.827} C_VEL
LIN {X 0,Y 580.308,Z 123.825,A -85,B 0,C 180,E1 -1791.644,E2 -1791.644} C_VEL
LIN {X 0,Y 580.312,Z 123.819,A -85,B 0,C 180,E1 -1794.44,E2 -1794.44} C_VEL
LIN {X 0,Y 580.344,Z 123.818,A -85,B 0,C 180,E1 -1797.918,E2 -1797.918} C_VEL
LIN {X 0,Y 580.344,Z 123.814,A -85,B 0,C 180,E1 -1800.694,E2 -1800.694} C_VEL
LIN {X 0,Y 580.321,Z 123.817,A -85,B 0,C 180,E1 -1802.777,E2 -1802.777} C_VEL
LIN {X 0,Y 580.328,Z 123.823,A -85,B 0,C 180,E1 -1805.56,E2 -1805.56} C_VEL
LIN {X 0,Y 580.308,Z 123.818,A -85,B 0,C 180,E1 -1808.356,E2 -1808.356} C_VEL
LIN {X 0,Y 580.304,Z 123.828,A -85,B 0,C 180,E1 -1811.191,E2 -1811.191} C_VEL
LIN {X 0,Y 580.31,Z 123.818,A -85,B 0,C 180,E1 -1814.017,E2 -1814.017} C_VEL
LIN {X 0,Y 580.292,Z 123.827,A -85,B 0,C 180,E1 -1816.906,E2 -1816.906} C_VEL
LIN {X 0,Y 580.284,Z 123.821,A -85,B 0,C 180,E1 -1819.823,E2 -1819.823} C_VEL
LIN {X 0,Y 580.259,Z 123.824,A -85,B 0,C 180,E1 -1822.053,E2 -1822.053} C_VEL
LIN {X 0,Y 580.289,Z 123.825,A -85,B 0,C 180,E1 -1825.08,E2 -1825.08} C_VEL
LIN {X 0,Y 580.292,Z 123.821,A -85,B 0,C 180,E1 -1827.857,E2 -1827.857} C_VEL
LIN {X 0,Y 580.274,Z 123.83,A -85,B 0,C 180,E1 -1830.692,E2 -1830.692} C_VEL
LIN {X 0,Y 580.285,Z 123.818,A -85,B 0,C 180,E1 -1833.313,E2 -1833.313} C_VEL
LIN {X 0,Y 580.246,Z 123.827,A -85,B 0,C 180,E1 -1835.756,E2 -1835.756} C_VEL
LIN {X 0,Y 580.288,Z 123.827,A -85,B 0,C 180,E1 -1838.146,E2 -1838.146} C_VEL
LIN {X 0,Y 580.298,Z 123.821,A -85,B 0,C 180,E1 -1840.843,E2 -1840.843} C_VEL
LIN {X 0,Y 580.281,Z 123.824,A -85,B 0,C 180,E1 -1843.658,E2 -1843.658} C_VEL
LIN {X 0,Y 580.275,Z 123.826,A -85,B 0,C 180,E1 -1846.61,E2 -1846.61} C_VEL
LIN {X 0,Y 580.3,Z 123.82,A -85,B 0,C 180,E1 -1849.156,E2 -1849.156} C_VEL
LIN {X 0,Y 580.291,Z 123.828,A -85,B 0,C 180,E1 -1851.927,E2 -1851.927} C_VEL
LIN {X 0,Y 580.251,Z 123.829,A -85,B 0,C 180,E1 -1854.453,E2 -1854.453} C_VEL
LIN {X 0,Y 580.291,Z 123.82,A -85,B 0,C 180,E1 -1856.975,E2 -1856.975} C_VEL
LIN {X 0,Y 580.297,Z 123.822,A -85,B 0,C 180,E1 -1859.425,E2 -1859.425} C_VEL
LIN {X 0,Y 580.298,Z 123.821,A -85,B 0,C 180,E1 -1862.141,E2 -1862.141} C_VEL
LIN {X 0,Y 580.349,Z 124.041,A -85,B 0,C 180,E1 -1864.802,E2 -1864.802} C_VEL
LIN {X 0,Y 581.262,Z 128.626,A -85,B 0,C 180,E1 -1865.439,E2 -1865.439} C_VEL
LIN {X 0,Y 581.077,Z 148.812,A -85,B 0,C 180,E1 -1867.979,E2 -1867.979} C_VEL
LIN {X 0,Y 580.855,Z 170.197,A -85,B 0,C 180,E1 -1870.611,E2 -1870.611} C_VEL
LIN {X 0,Y 581.878,Z 175.637,A -85,B 0,C 180,E1 -1870.74,E2 -1870.74} C_VEL
LIN {X 0,Y 581.541,Z 335.55,A -85,B 0,C 180,E1 -1872.782,E2 -1872.782} C_VEL
LIN {X 0,Y 581.429,Z 351.031,A -85,B 0,C 180,E1 -1873.118,E2 -1873.118} C_VEL
LIN {X 0,Y 581.28,Z 365.794,A -85,B 0,C 180,E1 -1873.583,E2 -1873.583} C_VEL
LIN {X 0,Y 581.127,Z 378.801,A -85,B 0,C 180,E1 -1874.12,E2 -1874.12} C_VEL
LIN {X 0,Y 580.947,Z 392.677,A -85,B 0,C 180,E1 -1874.834,E2 -1874.834} C_VEL
LIN {X 0,Y 580.783,Z 406.305,A -85,B 0,C 180,E1 -1875.7,E2 -1875.7} C_VEL
LIN {X 0,Y 580.608,Z 419.289,A -85,B 0,C 180,E1 -1876.704,E2 -1876.704} C_VEL
LIN {X 0,Y 580.479,Z 430.748,A -85,B 0,C 180,E1 -1877.768,E2 -1877.768} C_VEL
LIN {X 0,Y 580.307,Z 441.454,A -85,B 0,C 180,E1 -1878.954,E2 -1878.954} C_VEL
LIN {X 0,Y 580.268,Z 449.857,A -85,B 0,C 180,E1 -1880.061,E2 -1880.061} C_VEL
LIN {X 0,Y 580.215,Z 457.733,A -85,B 0,C 180,E1 -1881.291,E2 -1881.291} C_VEL
LIN {X 0,Y 580.13,Z 465.089,A -85,B 0,C 180,E1 -1882.692,E2 -1882.692} C_VEL
LIN {X 0,Y 580.132,Z 470.923,A -85,B 0,C 180,E1 -1884.09,E2 -1884.09} C_VEL
LIN {X 0,Y 580.041,Z 474.385,A -85,B 0,C 180,E1 -1885.135,E2 -1885.135} C_VEL
LIN {X 0,Y 580.105,Z 477.889,A -85,B 0,C 180,E1 -1886.527,E2 -1886.527} C_VEL
LIN {X 0,Y 580.039,Z 480.192,A -85,B 0,C 180,E1 -1887.917,E2 -1887.917} C_VEL
LIN {X 0,Y 580.036,Z 481.349,A -85,B 0,C 180,E1 -1889.306,E2 -1889.306} C_VEL
LIN {X 0,Y 580.036,Z 481.349,A -85,B 0,C 180,E1 -1890.694,E2 -1890.694} C_VEL
LIN {X 0,Y 580.039,Z 480.191,A -85,B 0,C 180,E1 -1892.083,E2 -1892.083} C_VEL
LIN {X 0,Y 580.105,Z 477.887,A -85,B 0,C 180,E1 -1893.473,E2 -1893.473} C_VEL
LIN {X 0,Y 580.041,Z 474.385,A -85,B 0,C 180,E1 -1894.865,E2 -1894.865} C_VEL
LIN {X 0,Y 580.093,Z 469.608,A -85,B 0,C 180,E1 -1896.26,E2 -1896.26} C_VEL
LIN {X 0,Y 580.165,Z 463.423,A -85,B 0,C 180,E1 -1897.658,E2 -1897.658} C_VEL
LIN {X 0,Y 580.207,Z 455.649,A -85,B 0,C 180,E1 -1899.06,E2 -1899.06} C_VEL
LIN {X 0,Y 580.308,Z 447.369,A -85,B 0,C 180,E1 -1900.29,E2 -1900.29} C_VEL
LIN {X 0,Y 580.383,Z 437.395,A -85,B 0,C 180,E1 -1901.525,E2 -1901.525} C_VEL
LIN {X 0,Y 580.541,Z 427.189,A -85,B 0,C 180,E1 -1902.586,E2 -1902.586} C_VEL
LIN {X 0,Y 580.677,Z 415.019,A -85,B 0,C 180,E1 -1903.651,E2 -1903.651} C_VEL
LIN {X 0,Y 580.874,Z 401.529,A -85,B 0,C 180,E1 -1904.625,E2 -1904.625} C_VEL
LIN {X 0,Y 581.013,Z 387.87,A -85,B 0,C 180,E1 -1905.433,E2 -1905.433} C_VEL
LIN {X 0,Y 581.208,Z 373.798,A -85,B 0,C 180,E1 -1906.103,E2 -1906.103} C_VEL
LIN {X 0,Y 581.368,Z 359.303,A -85,B 0,C 180,E1 -1906.64,E2 -1906.64} C_VEL
LIN {X 0,Y 581.498,Z 344.116,A -85,B 0,C 180,E1 -1907.051,E2 -1907.051} C_VEL
LIN {X 0,Y 581.563,Z 328.301,A -85,B 0,C 180,E1 -1907.326,E2 -1907.326} C_VEL
LIN {X 0,Y 581.851,Z 175.41,A -85,B 0,C 180,E1 -1909.264,E2 -1909.264} C_VEL
LIN {X 0,Y 580.88,Z 170.338,A -85,B 0,C 180,E1 -1909.38,E2 -1909.38} C_VEL
LIN {X 0,Y 581.077,Z 148.812,A -85,B 0,C 180,E1 -1912.021,E2 -1912.021} C_VEL
LIN {X 0,Y 581.285,Z 129.756,A -85,B 0,C 180,E1 -1914.416,E2 -1914.416} C_VEL
LIN {X 0,Y 580.35,Z 124.038,A -85,B 0,C 180,E1 -1915.198,E2 -1915.198} C_VEL
LIN {X 0,Y 580.298,Z 123.823,A -85,B 0,C 180,E1 -1918.186,E2 -1918.186} C_VEL
LIN {X 0,Y 580.285,Z 123.822,A -85,B 0,C 180,E1 -1920.695,E2 -1920.695} C_VEL
LIN {X 0,Y 580.304,Z 123.819,A -85,B 0,C 180,E1 -1923.316,E2 -1923.316} C_VEL
LIN {X 0,Y 580.246,Z 123.833,A -85,B 0,C 180,E1 -1925.756,E2 -1925.756} C_VEL
LIN {X 0,Y 580.29,Z 123.827,A -85,B 0,C 180,E1 -1928.146,E2 -1928.146} C_VEL
LIN {X 0,Y 580.3,Z 123.82,A -85,B 0,C 180,E1 -1930.843,E2 -1930.843} C_VEL
LIN {X 0,Y 580.274,Z 123.83,A -85,B 0,C 180,E1 -1933.658,E2 -1933.658} C_VEL
LIN {X 0,Y 580.279,Z 123.823,A -85,B 0,C 180,E1 -1936.609,E2 -1936.609} C_VEL
LIN {X 0,Y 580.298,Z 123.821,A -85,B 0,C 180,E1 -1939.157,E2 -1939.157} C_VEL
LIN {X 0,Y 580.289,Z 123.826,A -85,B 0,C 180,E1 -1941.927,E2 -1941.927} C_VEL
LIN {X 0,Y 580.251,Z 123.825,A -85,B 0,C 180,E1 -1944.453,E2 -1944.453} C_VEL
LIN {X 0,Y 580.29,Z 123.819,A -85,B 0,C 180,E1 -1946.975,E2 -1946.975} C_VEL
LIN {X 0,Y 580.288,Z 123.83,A -85,B 0,C 180,E1 -1949.425,E2 -1949.425} C_VEL
LIN {X 0,Y 580.292,Z 123.821,A -85,B 0,C 180,E1 -1952.143,E2 -1952.143} C_VEL
LIN {X 0,Y 580.322,Z 123.826,A -85,B 0,C 180,E1 -1955.27,E2 -1955.27} C_VEL
LIN {X 0,Y 580.268,Z 123.823,A -85,B 0,C 180,E1 -1957.947,E2 -1957.947} C_VEL
LIN {X 0,Y 580.296,Z 123.828,A -85,B 0,C 180,E1 -1960.913,E2 -1960.913} C_VEL
LIN {X 0,Y 580.263,Z 123.823,A -85,B 0,C 180,E1 -1963.825,E2 -1963.825} C_VEL
LIN {X 0,Y 580.267,Z 123.83,A -85,B 0,C 180,E1 -1966.696,E2 -1966.696} C_VEL
LIN {X 0,Y 580.308,Z 123.827,A -85,B 0,C 180,E1 -1968.827,E2 -1968.827} C_VEL
LIN {X 0,Y 580.309,Z 123.818,A -85,B 0,C 180,E1 -1971.644,E2 -1971.644} C_VEL
LIN {X 0,Y 580.33,Z 123.822,A -85,B 0,C 180,E1 -1974.44,E2 -1974.44} C_VEL
LIN {X 0,Y 580.342,Z 123.815,A -85,B 0,C 180,E1 -1977.918,E2 -1977.918} C_VEL
LIN {X 0,Y 580.358,Z 123.818,A -85,B 0,C 180,E1 -1980.694,E2 -1980.694} C_VEL
LIN {X 0,Y 580.327,Z 123.819,A -85,B 0,C 180,E1 -1982.777,E2 -1982.777} C_VEL
LIN {X 0,Y 580.314,Z 123.819,A -85,B 0,C 180,E1 -1985.56,E2 -1985.56} C_VEL
LIN {X 0,Y 580.324,Z 123.824,A -85,B 0,C 180,E1 -1988.356,E2 -1988.356} C_VEL
LIN {X 0,Y 580.303,Z 123.819,A -85,B 0,C 180,E1 -1991.191,E2 -1991.191} C_VEL
LIN {X 0,Y 580.314,Z 123.826,A -85,B 0,C 180,E1 -1994.017,E2 -1994.017} C_VEL
LIN {X 0,Y 580.251,Z 123.826,A -85,B 0,C 180,E1 -1996.899,E2 -1996.899} C_VEL
LIN {X 0,Y 580.278,Z 123.83,A -85,B 0,C 180,E1 -1999.823,E2 -1999.823} C_VEL
LIN {X 0,Y 580.284,Z 123.823,A -85,B 0,C 180,E1 -2001.316,E2 -2001.316} C_VEL
LIN {X 0,Y 579.576,Z 123.92,A -85,B 0,C 180,E1 -2001.895,E2 -2001.895} C_VEL
LIN {X 0,Y 576.692,Z 124.274,A -85,B 0,C 180,E1 -2002.835,E2 -2002.835} C_VEL
LIN {X 0,Y 574.291,Z 124.574,A -85,B 0,C 180,E1 -2003.591,E2 -2003.591} C_VEL
LIN {X 0,Y 573.281,Z 124.697,A -85,B 0,C 180,E1 -2004.175,E2 -2004.175} C_VEL
LIN {X 0,Y 573.208,Z 124.704,A -85,B 0,C 180,E1 -2004.372,E2 -2004.372} C_VEL
LIN {X 0,Y 573.199,Z 124.705,A -85,B 0,C 180,E1 -2006.979,E2 -2006.979} C_VEL
LIN {X 0,Y 573.222,Z 124.708,A -85,B 0,C 180,E1 -2009.483,E2 -2009.483} C_VEL
LIN {X 0,Y 573.237,Z 124.694,A -85,B 0,C 180,E1 -2012.226,E2 -2012.226} C_VEL
LIN {X 0,Y 573.222,Z 124.701,A -85,B 0,C 180,E1 -2014.769,E2 -2014.769} C_VEL
LIN {X 0,Y 573.226,Z 124.704,A -85,B 0,C 180,E1 -2017.808,E2 -2017.808} C_VEL
LIN {X 0,Y 573.246,Z 124.693,A -85,B 0,C 180,E1 -2020.525,E2 -2020.525} C_VEL
LIN {X 0,Y 573.206,Z 124.707,A -85,B 0,C 180,E1 -2023.665,E2 -2023.665} C_VEL
LIN {X 0,Y 573.2,Z 124.704,A -85,B 0,C 180,E1 -2026.637,E2 -2026.637} C_VEL
LIN {X 0,Y 573.246,Z 124.701,A -85,B 0,C 180,E1 -2029.475,E2 -2029.475} C_VEL
LIN {X 0,Y 573.225,Z 124.702,A -85,B 0,C 180,E1 -2032.192,E2 -2032.192} C_VEL
LIN {X 0,Y 573.218,Z 124.708,A -85,B 0,C 180,E1 -2035.231,E2 -2035.231} C_VEL
LIN {X 0,Y 573.236,Z 124.701,A -85,B 0,C 180,E1 -2037.775,E2 -2037.775} C_VEL
LIN {X 0,Y 573.214,Z 124.705,A -85,B 0,C 180,E1 -2040.631,E2 -2040.631} C_VEL
LIN {X 0,Y 573.198,Z 124.706,A -85,B 0,C 180,E1 -2043.516,E2 -2043.516} C_VEL
LIN {X 0,Y 573.243,Z 124.853,A -85,B 0,C 180,E1 -2045.606,E2 -2045.606} C_VEL
LIN {X 0,Y 574.29,Z 130.599,A -85,B 0,C 180,E1 -2046.463,E2 -2046.463} C_VEL
LIN {X 0,Y 574.035,Z 149.859,A -85,B 0,C 180,E1 -2049.033,E2 -2049.033} C_VEL
LIN {X 0,Y 573.932,Z 160.695,A -85,B 0,C 180,E1 -2050.424,E2 -2050.424} C_VEL
LIN {X 0,Y 575.192,Z 167.234,A -85,B 0,C 180,E1 -2050.572,E2 -2050.572} C_VEL
LIN {X 0,Y 574.743,Z 326.161,A -85,B 0,C 180,E1 -2052.627,E2 -2052.627} C_VEL
LIN {X 0,Y 574.61,Z 341.745,A -85,B 0,C 180,E1 -2052.976,E2 -2052.976} C_VEL
LIN {X 0,Y 574.431,Z 357.062,A -85,B 0,C 180,E1 -2053.474,E2 -2053.474} C_VEL
LIN {X 0,Y 574.26,Z 371.722,A -85,B 0,C 180,E1 -2054.107,E2 -2054.107} C_VEL
LIN {X 0,Y 574.032,Z 385.036,A -85,B 0,C 180,E1 -2054.829,E2 -2054.829} C_VEL
LIN {X 0,Y 573.859,Z 398.555,A -85,B 0,C 180,E1 -2055.728,E2 -2055.728} C_VEL
LIN {X 0,Y 573.631,Z 410.882,A -85,B 0,C 180,E1 -2056.719,E2 -2056.719} C_VEL
LIN {X 0,Y 573.459,Z 422.079,A -85,B 0,C 180,E1 -2057.795,E2 -2057.795} C_VEL
LIN {X 0,Y 573.295,Z 431.582,A -85,B 0,C 180,E1 -2058.877,E2 -2058.877} C_VEL
LIN {X 0,Y 573.203,Z 440.775,A -85,B 0,C 180,E1 -2060.116,E2 -2060.116} C_VEL
LIN {X 0,Y 573.134,Z 448.484,A -85,B 0,C 180,E1 -2061.361,E2 -2061.361} C_VEL
LIN {X 0,Y 573.075,Z 454.883,A -85,B 0,C 180,E1 -2062.602,E2 -2062.602} C_VEL
LIN {X 0,Y 573.042,Z 460.767,A -85,B 0,C 180,E1 -2064.016,E2 -2064.016} C_VEL
LIN {X 0,Y 572.949,Z 464.251,A -85,B 0,C 180,E1 -2065.074,E2 -2065.074} C_VEL
LIN {X 0,Y 573.004,Z 467.794,A -85,B 0,C 180,E1 -2066.484,E2 -2066.484} C_VEL
LIN {X 0,Y 572.938,Z 470.139,A -85,B 0,C 180,E1 -2067.891,E2 -2067.891} C_VEL
LIN {X 0,Y 572.936,Z 471.337,A -85,B 0,C 180,E1 -2069.297,E2 -2069.297} C_VEL
LIN {X 0,Y 572.937,Z 471.359,A -85,B 0,C 180,E1 -2070.703,E2 -2070.703} C_VEL
LIN {X 0,Y 572.939,Z 470.243,A -85,B 0,C 180,E1 -2072.109,E2 -2072.109} C_VEL
LIN {X 0,Y 573.006,Z 467.981,A -85,B 0,C 180,E1 -2073.516,E2 -2073.516} C_VEL
LIN {X 0,Y 572.949,Z 464.521,A -85,B 0,C 180,E1 -2074.926,E2 -2074.926} C_VEL
LIN {X 0,Y 573.007,Z 459.787,A -85,B 0,C 180,E1 -2076.338,E2 -2076.338} C_VEL
LIN {X 0,Y 573.094,Z 453.653,A -85,B 0,C 180,E1 -2077.753,E2 -2077.753} C_VEL
LIN {X 0,Y 573.134,Z 445.932,A -85,B 0,C 180,E1 -2079.173,E2 -2079.173} C_VEL
LIN {X 0,Y 573.265,Z 437.693,A -85,B 0,C 180,E1 -2080.418,E2 -2080.418} C_VEL
LIN {X 0,Y 573.354,Z 427.784,A -85,B 0,C 180,E1 -2081.669,E2 -2081.669} C_VEL
LIN {X 0,Y 573.534,Z 417.632,A -85,B 0,C 180,E1 -2082.743,E2 -2082.743} C_VEL
LIN {X 0,Y 573.722,Z 405.551,A -85,B 0,C 180,E1 -2083.82,E2 -2083.82} C_VEL
LIN {X 0,Y 573.919,Z 392.594,A -85,B 0,C 180,E1 -2084.78,E2 -2084.78} C_VEL
LIN {X 0,Y 574.136,Z 378.713,A -85,B 0,C 180,E1 -2085.623,E2 -2085.623} C_VEL
LIN {X 0,Y 574.356,Z 363.781,A -85,B 0,C 180,E1 -2086.346,E2 -2086.346} C_VEL
LIN {X 0,Y 574.548,Z 349.265,A -85,B 0,C 180,E1 -2086.889,E2 -2086.889} C_VEL
LIN {X 0,Y 574.687,Z 333.681,A -85,B 0,C 180,E1 -2087.314,E2 -2087.314} C_VEL
LIN {X 0,Y 574.799,Z 317.452,A -85,B 0,C 180,E1 -2087.592,E2 -2087.592} C_VEL
LIN {X 0,Y 575.112,Z 166.731,A -85,B 0,C 180,E1 -2089.527,E2 -2089.527} C_VEL
LIN {X 0,Y 573.941,Z 160.719,A -85,B 0,C 180,E1 -2089.664,E2 -2089.664} C_VEL
LIN {X 0,Y 574.147,Z 141.917,A -85,B 0,C 180,E1 -2092.111,E2 -2092.111} C_VEL
LIN {X 0,Y 574.298,Z 130.317,A -85,B 0,C 180,E1 -2093.665,E2 -2093.665} C_VEL
LIN {X 0,Y 573.219,Z 124.83,A -85,B 0,C 180,E1 -2094.492,E2 -2094.492} C_VEL
LIN {X 0,Y 573.182,Z 124.708,A -85,B 0,C 180,E1 -2096.98,E2 -2096.98} C_VEL
LIN {X 0,Y 573.195,Z 124.706,A -85,B 0,C 180,E1 -2099.479,E2 -2099.479} C_VEL
LIN {X 0,Y 573.228,Z 124.702,A -85,B 0,C 180,E1 -2102.224,E2 -2102.224} C_VEL
LIN {X 0,Y 573.215,Z 124.707,A -85,B 0,C 180,E1 -2104.768,E2 -2104.768} C_VEL
LIN {X 0,Y 573.22,Z 124.703,A -85,B 0,C 180,E1 -2107.809,E2 -2107.809} C_VEL
LIN {X 0,Y 573.211,Z 124.704,A -85,B 0,C 180,E1 -2110.528,E2 -2110.528} C_VEL
LIN {X 0,Y 573.199,Z 124.705,A -85,B 0,C 180,E1 -2113.363,E2 -2113.363} C_VEL
LIN {X 0,Y 573.206,Z 124.706,A -85,B 0,C 180,E1 -2116.335,E2 -2116.335} C_VEL
LIN {X 0,Y 573.229,Z 124.696,A -85,B 0,C 180,E1 -2119.477,E2 -2119.477} C_VEL
LIN {X 0,Y 573.222,Z 124.703,A -85,B 0,C 180,E1 -2122.191,E2 -2122.191} C_VEL
LIN {X 0,Y 573.22,Z 124.702,A -85,B 0,C 180,E1 -2125.231,E2 -2125.231} C_VEL
LIN {X 0,Y 573.237,Z 124.694,A -85,B 0,C 180,E1 -2127.775,E2 -2127.775} C_VEL
LIN {X 0,Y 573.239,Z 124.705,A -85,B 0,C 180,E1 -2130.633,E2 -2130.633} C_VEL
LIN {X 0,Y 573.21,Z 124.703,A -85,B 0,C 180,E1 -2133.514,E2 -2133.514} C_VEL
LIN {X 0,Y 573.2,Z 124.711,A -85,B 0,C 180,E1 -2136.133,E2 -2136.133} C_VEL
LIN {X 0,Y 573.237,Z 124.701,A -85,B 0,C 180,E1 -2138.714,E2 -2138.714} C_VEL
LIN {X 0,Y 573.201,Z 124.704,A -85,B 0,C 180,E1 -2141.41,E2 -2141.41} C_VEL
LIN {X 0,Y 573.213,Z 124.705,A -85,B 0,C 180,E1 -2144.351,E2 -2144.351} C_VEL
LIN {X 0,Y 573.211,Z 124.704,A -85,B 0,C 180,E1 -2146.529,E2 -2146.529} C_VEL
LIN {X 0,Y 573.263,Z 124.7,A -85,B 0,C 180,E1 -2149.403,E2 -2149.403} C_VEL
LIN {X 0,Y 573.262,Z 124.698,A -85,B 0,C 180,E1 -2152.25,E2 -2152.25} C_VEL
LIN {X 0,Y 573.292,Z 124.694,A -85,B 0,C 180,E1 -2155.077,E2 -2155.077} C_VEL
LIN {X 0,Y 573.314,Z 124.694,A -85,B 0,C 180,E1 -2157.892,E2 -2157.892} C_VEL
LIN {X 0,Y 573.317,Z 124.69,A -85,B 0,C 180,E1 -2160.702,E2 -2160.702} C_VEL
LIN {X 0,Y 573.289,Z 124.693,A -85,B 0,C 180,E1 -2162.811,E2 -2162.811} C_VEL
LIN {X 0,Y 573.295,Z 124.698,A -85,B 0,C 180,E1 -2165.628,E2 -2165.628} C_VEL
LIN {X 0,Y 573.252,Z 124.697,A -85,B 0,C 180,E1 -2168.46,E2 -2168.46} C_VEL
LIN {X 0,Y 573.275,Z 124.704,A -85,B 0,C 180,E1 -2171.312,E2 -2171.312} C_VEL
LIN {X 0,Y 573.265,Z 124.696,A -85,B 0,C 180,E1 -2174.417,E2 -2174.417} C_VEL
LIN {X 0,Y 573.249,Z 124.707,A -85,B 0,C 180,E1 -2177.112,E2 -2177.112} C_VEL
LIN {X 0,Y 573.239,Z 124.699,A -85,B 0,C 180,E1 -2180.077,E2 -2180.077} C_VEL
LIN {X 0,Y 573.226,Z 124.702,A -85,B 0,C 180,E1 -2182.338,E2 -2182.338} C_VEL
LIN {X 0,Y 573.241,Z 124.699,A -85,B 0,C 180,E1 -2185.411,E2 -2185.411} C_VEL
LIN {X 0,Y 573.247,Z 124.699,A -85,B 0,C 180,E1 -2188.028,E2 -2188.028} C_VEL
LIN {X 0,Y 573.237,Z 124.702,A -85,B 0,C 180,E1 -2190.177,E2 -2190.177} C_VEL
LIN {X 0,Y 573.254,Z 124.699,A -85,B 0,C 180,E1 -2192.645,E2 -2192.645} C_VEL
LIN {X 0,Y 573.207,Z 124.704,A -85,B 0,C 180,E1 -2195.188,E2 -2195.188} C_VEL
LIN {X 0,Y 573.235,Z 124.701,A -85,B 0,C 180,E1 -2197.807,E2 -2197.807} C_VEL
LIN {X 0,Y 573.246,Z 124.703,A -85,B 0,C 180,E1 -2200.525,E2 -2200.525} C_VEL
LIN {X 0,Y 573.242,Z 124.7,A -85,B 0,C 180,E1 -2203.359,E2 -2203.359} C_VEL
LIN {X 0,Y 573.24,Z 124.706,A -85,B 0,C 180,E1 -2206.331,E2 -2206.331} C_VEL
LIN {X 0,Y 573.231,Z 124.704,A -85,B 0,C 180,E1 -2208.543,E2 -2208.543} C_VEL
LIN {X 0,Y 573.25,Z 124.698,A -85,B 0,C 180,E1 -2211.299,E2 -2211.299} C_VEL
LIN {X 0,Y 573.213,Z 124.71,A -85,B 0,C 180,E1 -2214.018,E2 -2214.018} C_VEL
LIN {X 0,Y 573.27,Z 124.696,A -85,B 0,C 180,E1 -2216.518,E2 -2216.518} C_VEL
LIN {X 0,Y 573.229,Z 124.699,A -85,B 0,C 180,E1 -2219.118,E2 -2219.118} C_VEL
LIN {X 0,Y 573.238,Z 124.705,A -85,B 0,C 180,E1 -2221.435,E2 -2221.435} C_VEL
LIN {X 0,Y 573.247,Z 124.703,A -85,B 0,C 180,E1 -2224.395,E2 -2224.395} C_VEL
LIN {X 0,Y 573.296,Z 124.913,A -85,B 0,C 180,E1 -2224.592,E2 -2224.592} C_VEL
LIN {X 0,Y 574.436,Z 130.829,A -85,B 0,C 180,E1 -2225.419,E2 -2225.419} C_VEL
LIN {X 0,Y 574.191,Z 151.778,A -85,B 0,C 180,E1 -2228.08,E2 -2228.08} C_VEL
LIN {X 0,Y 573.963,Z 170.366,A -85,B 0,C 180,E1 -2230.378,E2 -2230.378} C_VEL
LIN {X 0,Y 575.197,Z 177.074,A -85,B 0,C 180,E1 -2230.526,E2 -2230.526} C_VEL
LIN {X 0,Y 574.758,Z 335.627,A -85,B 0,C 180,E1 -2232.573,E2 -2232.573} C_VEL
LIN {X 0,Y 574.643,Z 351.08,A -85,B 0,C 180,E1 -2232.914,E2 -2232.914} C_VEL
LIN {X 0,Y 574.464,Z 365.795,A -85,B 0,C 180,E1 -2233.383,E2 -2233.383} C_VEL
LIN {X 0,Y 574.266,Z 378.802,A -85,B 0,C 180,E1 -2233.925,E2 -2233.925} C_VEL
LIN {X 0,Y 574.055,Z 392.677,A -85,B 0,C 180,E1 -2234.648,E2 -2234.648} C_VEL
LIN {X 0,Y 573.847,Z 405.86,A -85,B 0,C 180,E1 -2235.493,E2 -2235.493} C_VEL
LIN {X 0,Y 573.656,Z 418.226,A -85,B 0,C 180,E1 -2236.449,E2 -2236.449} C_VEL
LIN {X 0,Y 573.511,Z 428.968,A -85,B 0,C 180,E1 -2237.437,E2 -2237.437} C_VEL
LIN {X 0,Y 573.349,Z 438.902,A -85,B 0,C 180,E1 -2238.51,E2 -2238.51} C_VEL
LIN {X 0,Y 573.256,Z 448.62,A -85,B 0,C 180,E1 -2239.76,E2 -2239.76} C_VEL
LIN {X 0,Y 573.135,Z 456.722,A -85,B 0,C 180,E1 -2241.005,E2 -2241.005} C_VEL
LIN {X 0,Y 573.093,Z 463.424,A -85,B 0,C 180,E1 -2242.247,E2 -2242.247} C_VEL
LIN {X 0,Y 573.015,Z 469.606,A -85,B 0,C 180,E1 -2243.662,E2 -2243.662} C_VEL
LIN {X 0,Y 572.951,Z 474.385,A -85,B 0,C 180,E1 -2245.074,E2 -2245.074} C_VEL
LIN {X 0,Y 573.005,Z 477.89,A -85,B 0,C 180,E1 -2246.484,E2 -2246.484} C_VEL
LIN {X 0,Y 572.938,Z 480.192,A -85,B 0,C 180,E1 -2247.891,E2 -2247.891} C_VEL
LIN {X 0,Y 572.936,Z 481.349,A -85,B 0,C 180,E1 -2249.297,E2 -2249.297} C_VEL
LIN {X 0,Y 572.936,Z 481.348,A -85,B 0,C 180,E1 -2250.703,E2 -2250.703} C_VEL
LIN {X 0,Y 572.938,Z 480.19,A -85,B 0,C 180,E1 -2252.109,E2 -2252.109} C_VEL
LIN {X 0,Y 573.005,Z 477.887,A -85,B 0,C 180,E1 -2253.516,E2 -2253.516} C_VEL
LIN {X 0,Y 572.951,Z 474.386,A -85,B 0,C 180,E1 -2254.926,E2 -2254.926} C_VEL
LIN {X 0,Y 573.014,Z 469.609,A -85,B 0,C 180,E1 -2256.337,E2 -2256.337} C_VEL
LIN {X 0,Y 573.093,Z 463.422,A -85,B 0,C 180,E1 -2257.753,E2 -2257.753} C_VEL
LIN {X 0,Y 573.135,Z 455.647,A -85,B 0,C 180,E1 -2259.173,E2 -2259.173} C_VEL
LIN {X 0,Y 573.27,Z 447.368,A -85,B 0,C 180,E1 -2260.418,E2 -2260.418} C_VEL
LIN {X 0,Y 573.386,Z 437.391,A -85,B 0,C 180,E1 -2261.668,E2 -2261.668} C_VEL
LIN {X 0,Y 573.568,Z 427.187,A -85,B 0,C 180,E1 -2262.742,E2 -2262.742} C_VEL
LIN {X 0,Y 573.742,Z 415.019,A -85,B 0,C 180,E1 -2263.819,E2 -2263.819} C_VEL
